# B&R Automation Studio project PT_KB_V01 (part 5)

#### vfdMain.st
```iecst
(* Glavni VFD orchestrator: kontrola, monitoring i dijagnostika po metodi rada. *)
FUNCTION_BLOCK vfdMain

	(* ---------------------------------------------------------------------- *)
	(* 1) Pristup centralnoj VFD strukturi preko prosledjene adrese            *)
	(* ---------------------------------------------------------------------- *)
	vfd_struct_data ACCESS addr_struct;

	(* ---------------------------------------------------------------------- *)
	(* 2) METOD_ENC_CANOPEN                                                     *)
	(* ---------------------------------------------------------------------- *)
	IF vfd_struct_data.settings.METOD_OF_CONTROL = METOD_ENC_CANOPEN THEN

		vfd_struct_data.status.act_power := UINT_TO_REAL(vfd_struct_data.mapping.CanOpen.r_power)/10.0;
		vfd_struct_data.status.act_current := UINT_TO_REAL(vfd_struct_data.mapping.CanOpen.r_current)/100.0;
		vfd_struct_data.status.act_torque := UINT_TO_REAL(vfd_struct_data.mapping.CanOpen.r_torque);
		vfd_struct_data.status.act_freq := UINT_TO_REAL(vfd_struct_data.mapping.CanOpen.r_freq)/100.0;
		vfd_struct_data.status.act_voltage := UINT_TO_REAL(vfd_struct_data.mapping.CanOpen.r_voltage);
		vfd_struct_data.status.act_velocity := UINT_TO_REAL(vfd_struct_data.mapping.CanOpen.r_velocity);

		IF vfd_struct_data.params.Freq > 100.0 THEN
			vfd_struct_data.params.Freq := 100.0;
		END_IF

		(* Skaliranje procentualnog zahteva frekvencije u raw CANopen opseg. *)
		vfd_struct_data.mapping.CanOpen.w_freq := REAL_TO_UINT((((vfd_struct_data.settings.MAX_Freq - vfd_struct_data.settings.MIN_Freq)/100.0)*vfd_struct_data.params.Freq - vfd_struct_data.settings.MIN_Freq)*100.0);
		vfd_struct_data.mapping.CanOpen.w_acc := REAL_TO_UINT(vfd_struct_data.params.Acc*10.0);
		vfd_struct_data.mapping.CanOpen.w_dec := REAL_TO_UINT(vfd_struct_data.params.Dec*10.0);

		fControlENC.cmd := vfd_struct_data.cmds;
		fControlENC.in_addr_CtrlWord := ADR(vfd_struct_data.mapping.CanOpen.CtrlWord);
		fControlENC.in_addr_StatusWord := ADR(vfd_struct_data.mapping.CanOpen.StatusWord);
		fControlENC.in_addr_r_CtrlWord := ADR(vfd_struct_data.mapping.CanOpen.r_CtrlWord);
		fControlENC();

		fStateENC.in_addr_StatusWord := ADR(vfd_struct_data.mapping.CanOpen.StatusWord);
		fStateENC();
		vfd_struct_data.states.state_word := fStateENC.out_State;

		IF NOT(vfd_struct_data.cmds.Enable) THEN
			state_case := ST_PWR_OFF;
		ELSE
			state_case := vfd_struct_data.states.state_word;
		END_IF;

		IF (vfd_struct_data.settings.HaveOverCurrentProtection) AND NOT(vfd_struct_data.mapping.CanOpenATV.r_OverCurrentProtect) THEN
			state_case := ST_CURRPROTECT;
			vfd_struct_data.states.OVERCURRENT_PROTECT := TRUE;
		ELSE
			vfd_struct_data.states.OVERCURRENT_PROTECT := FALSE;
		END_IF;

		Done := fControlENC.out_DONE;
		Busy := fControlENC.out_BUSY;
		errorID := vfd_struct_data.mapping.CanOpen.r_errorCode;

		(* Mapiranje internog state_case u bool state izlaze za HMI/SCADA. *)
		CASE state_case OF
			ST_PWR_OFF:
				vfd_struct_data.states.PWR_ON := FALSE;
				vfd_struct_data.states.READY := FALSE;
				vfd_struct_data.states.PREOPERATIONAL := FALSE;
				vfd_struct_data.states.RUN := FALSE;
				vfd_struct_data.states.STOPPING := FALSE;
				vfd_struct_data.states.STOPED := FALSE;
				vfd_struct_data.states.FAULT := FALSE;
				vfd_struct_data.states.ALARM := FALSE;
				vfd_struct_data.states.TUNING := FALSE;
				vfd_struct_data.states.JOG := FALSE;
			ST_READY:
				vfd_struct_data.states.PWR_ON := TRUE;
				vfd_struct_data.states.READY := TRUE;
				vfd_struct_data.states.PREOPERATIONAL := FALSE;
				vfd_struct_data.states.RUN := FALSE;
				vfd_struct_data.states.STOPPING := FALSE;
				vfd_struct_data.states.STOPED := FALSE;
				vfd_struct_data.states.FAULT := FALSE;
				vfd_struct_data.states.ALARM := FALSE;
				vfd_struct_data.states.TUNING := FALSE;
				vfd_struct_data.states.JOG := FALSE;
			ST_PREOPERATIONAL:
				vfd_struct_data.states.PWR_ON := TRUE;
				vfd_struct_data.states.READY := FALSE;
				vfd_struct_data.states.PREOPERATIONAL := TRUE;
				vfd_struct_data.states.RUN := FALSE;
				vfd_struct_data.states.STOPPING := FALSE;
				vfd_struct_data.states.STOPED := FALSE;
				vfd_struct_data.states.FAULT := FALSE;
				vfd_struct_data.states.ALARM := FALSE;
				vfd_struct_data.states.TUNING := FALSE;
				vfd_struct_data.states.JOG := FALSE;
			ST_RUN:
				vfd_struct_data.states.PWR_ON := TRUE;
				vfd_struct_data.states.READY := FALSE;
				vfd_struct_data.states.PREOPERATIONAL := FALSE;
				vfd_struct_data.states.RUN := TRUE;
				vfd_struct_data.states.STOPPING := FALSE;
				vfd_struct_data.states.STOPED := FALSE;
				vfd_struct_data.states.FAULT := FALSE;
				vfd_struct_data.states.ALARM := FALSE;
				vfd_struct_data.states.TUNING := FALSE;
				vfd_struct_data.states.JOG := FALSE;
			ST_STOPPING:
				vfd_struct_data.states.PWR_ON := TRUE;
				vfd_struct_data.states.READY := FALSE;
				vfd_struct_data.states.PREOPERATIONAL := FALSE;
				vfd_struct_data.states.RUN := FALSE;
				vfd_struct_data.states.STOPPING := TRUE;
				vfd_struct_data.states.STOPED := FALSE;
				vfd_struct_data.states.FAULT := FALSE;
				vfd_struct_data.states.ALARM := FALSE;
				vfd_struct_data.states.TUNING := FALSE;
				vfd_struct_data.states.JOG := FALSE;
			ST_STOPPED:
				vfd_struct_data.states.PWR_ON := TRUE;
				vfd_struct_data.states.READY := FALSE;
				vfd_struct_data.states.PREOPERATIONAL := FALSE;
				vfd_struct_data.states.RUN := FALSE;
				vfd_struct_data.states.STOPPING := FALSE;
				vfd_struct_data.states.STOPED := TRUE;
				vfd_struct_data.states.FAULT := FALSE;
				vfd_struct_data.states.ALARM := FALSE;
				vfd_struct_data.states.TUNING := FALSE;
				vfd_struct_data.states.JOG := FALSE;
			ST_FAULT:
				vfd_struct_data.states.PWR_ON := FALSE;
				vfd_struct_data.states.READY := FALSE;
				vfd_struct_data.states.PREOPERATIONAL := FALSE;
				vfd_struct_data.states.RUN := FALSE;
				vfd_struct_data.states.STOPPING := FALSE;
				vfd_struct_data.states.STOPED := FALSE;
				vfd_struct_data.states.FAULT := TRUE;
				vfd_struct_data.states.ALARM := FALSE;
				vfd_struct_data.states.TUNING := FALSE;
				vfd_struct_data.states.JOG := FALSE;
			ST_ALARM:
				vfd_struct_data.states.PWR_ON := TRUE;
				vfd_struct_data.states.READY := FALSE;
				vfd_struct_data.states.PREOPERATIONAL := FALSE;
				vfd_struct_data.states.RUN := FALSE;
				vfd_struct_data.states.STOPPING := FALSE;
				vfd_struct_data.states.STOPED := FALSE;
				vfd_struct_data.states.FAULT := FALSE;
				vfd_struct_data.states.ALARM := TRUE;
				vfd_struct_data.states.TUNING := FALSE;
				vfd_struct_data.states.JOG := FALSE;
			ST_TUNING:
				vfd_struct_data.states.PWR_ON := TRUE;
				vfd_struct_data.states.READY := FALSE;
				vfd_struct_data.states.PREOPERATIONAL := FALSE;
				vfd_struct_data.states.RUN := FALSE;
				vfd_struct_data.states.STOPPING := FALSE;
				vfd_struct_data.states.STOPED := FALSE;
				vfd_struct_data.states.FAULT := FALSE;
				vfd_struct_data.states.ALARM := FALSE;
				vfd_struct_data.states.TUNING := TRUE;
				vfd_struct_data.states.JOG := FALSE;
			ST_JOG:
				vfd_struct_data.states.PWR_ON := TRUE;
				vfd_struct_data.states.READY := FALSE;
				vfd_struct_data.states.PREOPERATIONAL := FALSE;
				vfd_struct_data.states.RUN := FALSE;
				vfd_struct_data.states.STOPPING := FALSE;
				vfd_struct_data.states.STOPED := FALSE;
				vfd_struct_data.states.FAULT := FALSE;
				vfd_struct_data.states.ALARM := FALSE;
				vfd_struct_data.states.TUNING := FALSE;
				vfd_struct_data.states.JOG := TRUE;
			ST_CURRPROTECT:
				vfd_struct_data.states.PWR_ON := FALSE;
				vfd_struct_data.states.READY := FALSE;
				vfd_struct_data.states.PREOPERATIONAL := FALSE;
				vfd_struct_data.states.RUN := FALSE;
				vfd_struct_data.states.STOPPING := FALSE;
				vfd_struct_data.states.STOPED := FALSE;
				vfd_struct_data.states.FAULT := FALSE;
				vfd_struct_data.states.ALARM := FALSE;
				vfd_struct_data.states.TUNING := FALSE;
				vfd_struct_data.states.JOG := FALSE;
				vfd_struct_data.states.OVERCURRENT_PROTECT := TRUE;
			ELSE
				vfd_struct_data.states.PWR_ON := TRUE;
				vfd_struct_data.states.READY := FALSE;
				vfd_struct_data.states.PREOPERATIONAL := FALSE;
				vfd_struct_data.states.RUN := FALSE;
				vfd_struct_data.states.STOPPING := FALSE;
				vfd_struct_data.states.STOPED := FALSE;
				vfd_struct_data.states.FAULT := FALSE;
				vfd_struct_data.states.ALARM := FALSE;
				vfd_struct_data.states.TUNING := FALSE;
				vfd_struct_data.states.JOG := FALSE;
		END_CASE;

	END_IF;

	(* ---------------------------------------------------------------------- *)
	(* 3) METOD_DIO                                                             *)
	(* ---------------------------------------------------------------------- *)
	IF vfd_struct_data.settings.METOD_OF_CONTROL = METOD_DIO THEN

		IF vfd_struct_data.cmds.Enable THEN

			(* Legacy ekvivalent skale: REAL_TO_INT((Freq)*32767.0/100.0). *)
			IF vfd_struct_data.params.Freq > 100.0 THEN
				vfd_struct_data.params.Freq := 100.0;
			END_IF

			vfd_struct_data.mapping.DIO.w_freq := REAL_TO_INT((32767.0/100.0)*vfd_struct_data.params.Freq);
			vfd_struct_data.mapping.DIO.w_run_fwd := vfd_struct_data.cmds.Run_fwd;
			vfd_struct_data.mapping.DIO.w_run_rev := vfd_struct_data.cmds.Run_rev;
			vfd_struct_data.mapping.DIO.w_jog_fwd := vfd_struct_data.cmds.Jog_fwd;
			vfd_struct_data.mapping.DIO.w_jog_rev := vfd_struct_data.cmds.Jog_rev;
			vfd_struct_data.mapping.DIO.w_Stop := vfd_struct_data.cmds.Stop;
			vfd_struct_data.mapping.DIO.w_faststop := vfd_struct_data.cmds.FastStop;

			vfd_struct_data.status.act_freq := (((vfd_struct_data.settings.MAX_Freq - vfd_struct_data.settings.MIN_Freq)/32767.0)*vfd_struct_data.mapping.DIO.r_freq - vfd_struct_data.settings.MIN_Freq)*100.0;

			(* Legacy ekvivalent citanja: REAL_TO_UINT((r_freq)*100.0/32767.0). *)
			state_case := ST_READY;
		ELSE
			vfd_struct_data.mapping.DIO.w_freq := 0;
			vfd_struct_data.mapping.DIO.w_run_fwd := FALSE;
			vfd_struct_data.mapping.DIO.w_run_rev := FALSE;
			vfd_struct_data.mapping.DIO.w_jog_fwd := FALSE;
			vfd_struct_data.mapping.DIO.w_jog_rev := FALSE;
			vfd_struct_data.mapping.DIO.w_Stop := FALSE;
			vfd_struct_data.mapping.DIO.w_faststop := FALSE;
			state_case := ST_PWR_OFF;
		END_IF

			vfd_struct_data.mapping.DIO.w_reset := vfd_struct_data.cmds.Reset;
		   IF NOT (vfd_struct_data.mapping.DIO.r_error) THEN
			   state_case := ST_FAULT;
		   END_IF

		IF (vfd_struct_data.settings.HaveOverCurrentProtection) AND NOT(vfd_struct_data.mapping.CanOpenATV.r_OverCurrentProtect) THEN
			state_case := ST_CURRPROTECT;
			vfd_struct_data.states.OVERCURRENT_PROTECT := TRUE;
		ELSE
			vfd_struct_data.states.OVERCURRENT_PROTECT := FALSE;
		END_IF;

		(* U DIO metodi koristi se isti izlazni model states.*)
		CASE state_case OF
			ST_PWR_OFF:
				vfd_struct_data.states.PWR_ON := FALSE;
				vfd_struct_data.states.READY := FALSE;
				vfd_struct_data.states.PREOPERATIONAL := FALSE;
				vfd_struct_data.states.RUN := FALSE;
				vfd_struct_data.states.STOPPING := FALSE;
				vfd_struct_data.states.STOPED := FALSE;
				vfd_struct_data.states.FAULT := FALSE;
				vfd_struct_data.states.ALARM := FALSE;
				vfd_struct_data.states.TUNING := FALSE;
				vfd_struct_data.states.JOG := FALSE;
			ST_READY:
				vfd_struct_data.states.PWR_ON := TRUE;
				vfd_struct_data.states.READY := TRUE;
				vfd_struct_data.states.PREOPERATIONAL := FALSE;
				vfd_struct_data.states.RUN := FALSE;
				vfd_struct_data.states.STOPPING := FALSE;
				vfd_struct_data.states.STOPED := FALSE;
				vfd_struct_data.states.FAULT := FALSE;
				vfd_struct_data.states.ALARM := FALSE;
				vfd_struct_data.states.TUNING := FALSE;
				vfd_struct_data.states.JOG := FALSE;
			ST_PREOPERATIONAL:
				vfd_struct_data.states.PWR_ON := TRUE;
				vfd_struct_data.states.READY := FALSE;
				vfd_struct_data.states.PREOPERATIONAL := TRUE;
				vfd_struct_data.states.RUN := FALSE;
				vfd_struct_data.states.STOPPING := FALSE;
				vfd_struct_data.states.STOPED := FALSE;
				vfd_struct_data.states.FAULT := FALSE;
				vfd_struct_data.states.ALARM := FALSE;
				vfd_struct_data.states.TUNING := FALSE;
				vfd_struct_data.states.JOG := FALSE;
			ST_RUN:
				vfd_struct_data.states.PWR_ON := TRUE;
				vfd_struct_data.states.READY := FALSE;
				vfd_struct_data.states.PREOPERATIONAL := FALSE;
				vfd_struct_data.states.RUN := TRUE;
				vfd_struct_data.states.STOPPING := FALSE;
				vfd_struct_data.states.STOPED := FALSE;
				vfd_struct_data.states.FAULT := FALSE;
				vfd_struct_data.states.ALARM := FALSE;
				vfd_struct_data.states.TUNING := FALSE;
				vfd_struct_data.states.JOG := FALSE;
			ST_STOPPING:
				vfd_struct_data.states.PWR_ON := TRUE;
				vfd_struct_data.states.READY := FALSE;
				vfd_struct_data.states.PREOPERATIONAL := FALSE;
				vfd_struct_data.states.RUN := FALSE;
				vfd_struct_data.states.STOPPING := TRUE;
				vfd_struct_data.states.STOPED := FALSE;
				vfd_struct_data.states.FAULT := FALSE;
				vfd_struct_data.states.ALARM := FALSE;
				vfd_struct_data.states.TUNING := FALSE;
				vfd_struct_data.states.JOG := FALSE;
			ST_STOPPED:
				vfd_struct_data.states.PWR_ON := TRUE;
				vfd_struct_data.states.READY := FALSE;
				vfd_struct_data.states.PREOPERATIONAL := FALSE;
				vfd_struct_data.states.RUN := FALSE;
				vfd_struct_data.states.STOPPING := FALSE;
				vfd_struct_data.states.STOPED := TRUE;
				vfd_struct_data.states.FAULT := FALSE;
				vfd_struct_data.states.ALARM := FALSE;
				vfd_struct_data.states.TUNING := FALSE;
				vfd_struct_data.states.JOG := FALSE;
			ST_FAULT:
				vfd_struct_data.states.PWR_ON := FALSE;
				vfd_struct_data.states.READY := FALSE;
				vfd_struct_data.states.PREOPERATIONAL := FALSE;
				vfd_struct_data.states.RUN := FALSE;
				vfd_struct_data.states.STOPPING := FALSE;
				vfd_struct_data.states.STOPED := FALSE;
				vfd_struct_data.states.FAULT := TRUE;
				vfd_struct_data.states.ALARM := FALSE;
				vfd_struct_data.states.TUNING := FALSE;
				vfd_struct_data.states.JOG := FALSE;
			ST_ALARM:
				vfd_struct_data.states.PWR_ON := TRUE;
				vfd_struct_data.states.READY := FALSE;
				vfd_struct_data.states.PREOPERATIONAL := FALSE;
				vfd_struct_data.states.RUN := FALSE;
				vfd_struct_data.states.STOPPING := FALSE;
				vfd_struct_data.states.STOPED := FALSE;
				vfd_struct_data.states.FAULT := FALSE;
				vfd_struct_data.states.ALARM := TRUE;
				vfd_struct_data.states.TUNING := FALSE;
				vfd_struct_data.states.JOG := FALSE;
			ST_TUNING:
				vfd_struct_data.states.PWR_ON := TRUE;
				vfd_struct_data.states.READY := FALSE;
				vfd_struct_data.states.PREOPERATIONAL := FALSE;
				vfd_struct_data.states.RUN := FALSE;
				vfd_struct_data.states.STOPPING := FALSE;
				vfd_struct_data.states.STOPED := FALSE;
				vfd_struct_data.states.FAULT := FALSE;
				vfd_struct_data.states.ALARM := FALSE;
				vfd_struct_data.states.TUNING := TRUE;
				vfd_struct_data.states.JOG := FALSE;
			ST_JOG:
				vfd_struct_data.states.PWR_ON := TRUE;
				vfd_struct_data.states.READY := FALSE;
				vfd_struct_data.states.PREOPERATIONAL := FALSE;
				vfd_struct_data.states.RUN := FALSE;
				vfd_struct_data.states.STOPPING := FALSE;
				vfd_struct_data.states.STOPED := FALSE;
				vfd_struct_data.states.FAULT := FALSE;
				vfd_struct_data.states.ALARM := FALSE;
				vfd_struct_data.states.TUNING := FALSE;
				vfd_struct_data.states.JOG := TRUE;
			ST_CURRPROTECT:
				vfd_struct_data.states.PWR_ON := FALSE;
				vfd_struct_data.states.READY := FALSE;
				vfd_struct_data.states.PREOPERATIONAL := FALSE;
				vfd_struct_data.states.RUN := FALSE;
				vfd_struct_data.states.STOPPING := FALSE;
				vfd_struct_data.states.STOPED := FALSE;
				vfd_struct_data.states.FAULT := FALSE;
				vfd_struct_data.states.ALARM := FALSE;
				vfd_struct_data.states.TUNING := FALSE;
				vfd_struct_data.states.JOG := FALSE;
				vfd_struct_data.states.OVERCURRENT_PROTECT := TRUE;
			ELSE
				vfd_struct_data.states.PWR_ON := TRUE;
				vfd_struct_data.states.READY := FALSE;
				vfd_struct_data.states.PREOPERATIONAL := FALSE;
				vfd_struct_data.states.RUN := FALSE;
				vfd_struct_data.states.STOPPING := FALSE;
				vfd_struct_data.states.STOPED := FALSE;
				vfd_struct_data.states.FAULT := FALSE;
				vfd_struct_data.states.ALARM := FALSE;
				vfd_struct_data.states.TUNING := FALSE;
				vfd_struct_data.states.JOG := FALSE;
		END_CASE;

	END_IF;

	(* ---------------------------------------------------------------------- *)
	(* 4) METOD_DIO_CANOPEN                                                     *)
	(* ---------------------------------------------------------------------- *)
	IF vfd_struct_data.settings.METOD_OF_CONTROL = METOD_DIO_CANOPEN THEN

		IF vfd_struct_data.cmds.Enable THEN

			IF vfd_struct_data.params.Freq > 100.0 THEN
				vfd_struct_data.params.Freq := 100.0;
			END_IF

			vfd_struct_data.mapping.DIO.w_freq := REAL_TO_INT((32767.0/100.0)*vfd_struct_data.params.Freq);

			(* Legacy alternativa skale (ne koristi se u aktivnoj logici). *)
			vfd_struct_data.mapping.DIO.w_run_fwd := vfd_struct_data.cmds.Run_fwd;
			vfd_struct_data.mapping.DIO.w_run_rev := vfd_struct_data.cmds.Run_rev;
			vfd_struct_data.mapping.DIO.w_jog_fwd := vfd_struct_data.cmds.Jog_fwd;
			vfd_struct_data.mapping.DIO.w_jog_rev := vfd_struct_data.cmds.Jog_rev;
			vfd_struct_data.mapping.DIO.w_Stop := vfd_struct_data.cmds.Stop;
			vfd_struct_data.mapping.DIO.w_faststop := vfd_struct_data.cmds.FastStop;
			(* Legacy ekvivalent citanja: REAL_TO_UINT((r_freq)*100.0/32767.0). *)
		ELSE
			vfd_struct_data.mapping.DIO.w_freq := 0;
			vfd_struct_data.mapping.DIO.w_run_fwd := FALSE;
			vfd_struct_data.mapping.DIO.w_run_rev := FALSE;
			vfd_struct_data.mapping.DIO.w_jog_fwd := FALSE;
			vfd_struct_data.mapping.DIO.w_jog_rev := FALSE;
			vfd_struct_data.mapping.DIO.w_Stop := FALSE;
			vfd_struct_data.mapping.DIO.w_faststop := FALSE;

		END_IF

		vfd_struct_data.mapping.DIO.w_reset := vfd_struct_data.cmds.Reset;

		vfd_struct_data.status.act_power := UINT_TO_REAL(vfd_struct_data.mapping.CanOpen.r_power)/10.0;
		vfd_struct_data.status.act_current := UINT_TO_REAL(vfd_struct_data.mapping.CanOpen.r_current)/100.0;
		vfd_struct_data.status.act_torque := UINT_TO_REAL(vfd_struct_data.mapping.CanOpen.r_torque);
		vfd_struct_data.status.act_freq := UINT_TO_REAL(vfd_struct_data.mapping.CanOpen.r_freq)/100.0;
		vfd_struct_data.status.act_voltage := UINT_TO_REAL(vfd_struct_data.mapping.CanOpen.r_voltage);
		vfd_struct_data.status.act_velocity := UINT_TO_REAL(vfd_struct_data.mapping.CanOpen.r_velocity);

		vfd_struct_data.mapping.CanOpen.w_acc := REAL_TO_UINT(vfd_struct_data.params.Acc*10.0);
		vfd_struct_data.mapping.CanOpen.w_dec := REAL_TO_UINT(vfd_struct_data.params.Dec*10.0);

		fStateENC.in_addr_StatusWord := ADR(vfd_struct_data.mapping.CanOpen.StatusWord);
		fStateENC();
		vfd_struct_data.states.state_word := fStateENC.out_State;

		IF NOT(vfd_struct_data.cmds.Enable) THEN
			state_case := ST_PWR_OFF;
		ELSE
			state_case := vfd_struct_data.states.state_word;
		END_IF;

		IF (vfd_struct_data.settings.HaveOverCurrentProtection) AND NOT(vfd_struct_data.mapping.CanOpenATV.r_OverCurrentProtect) THEN
			state_case := ST_CURRPROTECT;
			vfd_struct_data.states.OVERCURRENT_PROTECT := TRUE;
		ELSE
			vfd_struct_data.states.OVERCURRENT_PROTECT := FALSE;
		END_IF;

		(* U kombinovanoj metodi Done/Busy se ne preuzimaju iz ENC control FB-a. *)
		errorID := vfd_struct_data.mapping.CanOpen.r_errorCode;

		(* Kombinovana metoda: komande kroz DIO, status kroz CANopen. *)
		CASE state_case OF
			ST_PWR_OFF:
				vfd_struct_data.states.PWR_ON := FALSE;
				vfd_struct_data.states.READY := FALSE;
				vfd_struct_data.states.PREOPERATIONAL := FALSE;
				vfd_struct_data.states.RUN := FALSE;
				vfd_struct_data.states.STOPPING := FALSE;
				vfd_struct_data.states.STOPED := FALSE;
				vfd_struct_data.states.FAULT := FALSE;
				vfd_struct_data.states.ALARM := FALSE;
				vfd_struct_data.states.TUNING := FALSE;
				vfd_struct_data.states.JOG := FALSE;
			ST_READY:
				vfd_struct_data.states.PWR_ON := TRUE;
				vfd_struct_data.states.READY := TRUE;
				vfd_struct_data.states.PREOPERATIONAL := FALSE;
				vfd_struct_data.states.RUN := FALSE;
				vfd_struct_data.states.STOPPING := FALSE;
				vfd_struct_data.states.STOPED := FALSE;
				vfd_struct_data.states.FAULT := FALSE;
				vfd_struct_data.states.ALARM := FALSE;
				vfd_struct_data.states.TUNING := FALSE;
				vfd_struct_data.states.JOG := FALSE;
			ST_PREOPERATIONAL:
				vfd_struct_data.states.PWR_ON := TRUE;
				vfd_struct_data.states.READY := FALSE;
				vfd_struct_data.states.PREOPERATIONAL := TRUE;
				vfd_struct_data.states.RUN := FALSE;
				vfd_struct_data.states.STOPPING := FALSE;
				vfd_struct_data.states.STOPED := FALSE;
				vfd_struct_data.states.FAULT := FALSE;
				vfd_struct_data.states.ALARM := FALSE;
				vfd_struct_data.states.TUNING := FALSE;
				vfd_struct_data.states.JOG := FALSE;
			ST_RUN:
				vfd_struct_data.states.PWR_ON := TRUE;
				vfd_struct_data.states.READY := FALSE;
				vfd_struct_data.states.PREOPERATIONAL := FALSE;
				vfd_struct_data.states.RUN := TRUE;
				vfd_struct_data.states.STOPPING := FALSE;
				vfd_struct_data.states.STOPED := FALSE;
				vfd_struct_data.states.FAULT := FALSE;
				vfd_struct_data.states.ALARM := FALSE;
				vfd_struct_data.states.TUNING := FALSE;
				vfd_struct_data.states.JOG := FALSE;
			ST_STOPPING:
				vfd_struct_data.states.PWR_ON := TRUE;
				vfd_struct_data.states.READY := FALSE;
				vfd_struct_data.states.PREOPERATIONAL := FALSE;
				vfd_struct_data.states.RUN := FALSE;
				vfd_struct_data.states.STOPPING := TRUE;
				vfd_struct_data.states.STOPED := FALSE;
				vfd_struct_data.states.FAULT := FALSE;
				vfd_struct_data.states.ALARM := FALSE;
				vfd_struct_data.states.TUNING := FALSE;
				vfd_struct_data.states.JOG := FALSE;
			ST_STOPPED:
				vfd_struct_data.states.PWR_ON := TRUE;
				vfd_struct_data.states.READY := FALSE;
				vfd_struct_data.states.PREOPERATIONAL := FALSE;
				vfd_struct_data.states.RUN := FALSE;
				vfd_struct_data.states.STOPPING := FALSE;
				vfd_struct_data.states.STOPED := TRUE;
				vfd_struct_data.states.FAULT := FALSE;
				vfd_struct_data.states.ALARM := FALSE;
				vfd_struct_data.states.TUNING := FALSE;
				vfd_struct_data.states.JOG := FALSE;
			ST_FAULT:
				vfd_struct_data.states.PWR_ON := FALSE;
				vfd_struct_data.states.READY := FALSE;
				vfd_struct_data.states.PREOPERATIONAL := FALSE;
				vfd_struct_data.states.RUN := FALSE;
				vfd_struct_data.states.STOPPING := FALSE;
				vfd_struct_data.states.STOPED := FALSE;
				vfd_struct_data.states.FAULT := TRUE;
				vfd_struct_data.states.ALARM := FALSE;
				vfd_struct_data.states.TUNING := FALSE;
				vfd_struct_data.states.JOG := FALSE;
			ST_ALARM:
				vfd_struct_data.states.PWR_ON := TRUE;
				vfd_struct_data.states.READY := FALSE;
				vfd_struct_data.states.PREOPERATIONAL := FALSE;
				vfd_struct_data.states.RUN := FALSE;
				vfd_struct_data.states.STOPPING := FALSE;
				vfd_struct_data.states.STOPED := FALSE;
				vfd_struct_data.states.FAULT := FALSE;
				vfd_struct_data.states.ALARM := TRUE;
				vfd_struct_data.states.TUNING := FALSE;
				vfd_struct_data.states.JOG := FALSE;
			ST_TUNING:
				vfd_struct_data.states.PWR_ON := TRUE;
				vfd_struct_data.states.READY := FALSE;
				vfd_struct_data.states.PREOPERATIONAL := FALSE;
				vfd_struct_data.states.RUN := FALSE;
				vfd_struct_data.states.STOPPING := FALSE;
				vfd_struct_data.states.STOPED := FALSE;
				vfd_struct_data.states.FAULT := FALSE;
				vfd_struct_data.states.ALARM := FALSE;
				vfd_struct_data.states.TUNING := TRUE;
				vfd_struct_data.states.JOG := FALSE;
			ST_JOG:
				vfd_struct_data.states.PWR_ON := TRUE;
				vfd_struct_data.states.READY := FALSE;
				vfd_struct_data.states.PREOPERATIONAL := FALSE;
				vfd_struct_data.states.RUN := FALSE;
				vfd_struct_data.states.STOPPING := FALSE;
				vfd_struct_data.states.STOPED := FALSE;
				vfd_struct_data.states.FAULT := FALSE;
				vfd_struct_data.states.ALARM := FALSE;
				vfd_struct_data.states.TUNING := FALSE;
				vfd_struct_data.states.JOG := TRUE;
			ST_CURRPROTECT:
				vfd_struct_data.states.PWR_ON := FALSE;
				vfd_struct_data.states.READY := FALSE;
				vfd_struct_data.states.PREOPERATIONAL := FALSE;
				vfd_struct_data.states.RUN := FALSE;
				vfd_struct_data.states.STOPPING := FALSE;
				vfd_struct_data.states.STOPED := FALSE;
				vfd_struct_data.states.FAULT := FALSE;
				vfd_struct_data.states.ALARM := FALSE;
				vfd_struct_data.states.TUNING := FALSE;
				vfd_struct_data.states.JOG := FALSE;
				vfd_struct_data.states.OVERCURRENT_PROTECT := TRUE;
			ELSE
				vfd_struct_data.states.PWR_ON := TRUE;
				vfd_struct_data.states.READY := FALSE;
				vfd_struct_data.states.PREOPERATIONAL := FALSE;
				vfd_struct_data.states.RUN := FALSE;
				vfd_struct_data.states.STOPPING := FALSE;
				vfd_struct_data.states.STOPED := FALSE;
				vfd_struct_data.states.FAULT := FALSE;
				vfd_struct_data.states.ALARM := FALSE;
				vfd_struct_data.states.TUNING := FALSE;
				vfd_struct_data.states.JOG := FALSE;
		END_CASE;

	END_IF;

	(* ---------------------------------------------------------------------- *)
	(* 5) METOD_ATV_CANOPEN                                                     *)
	(* ---------------------------------------------------------------------- *)
	IF vfd_struct_data.settings.METOD_OF_CONTROL = METOD_ATV_CANOPEN THEN

		vfd_struct_data.status.act_power := INT_TO_REAL(vfd_struct_data.mapping.CanOpenATV.r_power)*vfd_struct_data.settings.RatedMotorPower/100.0;
		vfd_struct_data.status.act_current := UINT_TO_REAL(vfd_struct_data.mapping.CanOpenATV.r_current)/10.0;
		vfd_struct_data.status.act_torque := INT_TO_REAL(vfd_struct_data.mapping.CanOpenATV.r_torque);
		vfd_struct_data.status.act_freq := INT_TO_REAL(vfd_struct_data.mapping.CanOpenATV.r_freq)/100.0;
		vfd_struct_data.status.act_voltage := UINT_TO_REAL(vfd_struct_data.mapping.CanOpenATV.r_voltage);
		vfd_struct_data.status.act_velocity := INT_TO_REAL(vfd_struct_data.mapping.CanOpenATV.ControlEffort);

		vfd_struct_data.mapping.CanOpenATV.w_acc := REAL_TO_UINT(vfd_struct_data.params.Acc*10.0);
		vfd_struct_data.mapping.CanOpenATV.w_dec := REAL_TO_UINT(vfd_struct_data.params.Dec*10.0);

		fStateATV.in_addr_StatusWord := ADR(vfd_struct_data.mapping.CanOpenATV.StatusWord);
		fStateATV();
		vfd_struct_data.states.state_word := fStateATV.out_State;

		fControlATV.cmd := vfd_struct_data.cmds;
		fControlATV.in_addr_CtrlWord := ADR(vfd_struct_data.mapping.CanOpenATV.CtrlWord);
		fControlATV.DC_BUS_STATE := fStateATV.DC_BUS_ON;
		fControlATV.StatusWord := fStateATV.out_State;

		IF vfd_struct_data.params.Freq > 100.0 THEN
			vfd_struct_data.params.Freq := 100.0;
		END_IF

		(* Konverzija procentualnog SP u ATV velocity zahtev. *)
		fControlATV.in_set_freq := REAL_TO_INT(vfd_struct_data.params.Freq*(vfd_struct_data.settings.MAX_Velocity)/100.0);

		fControlATV();
		vfd_struct_data.mapping.CanOpenATV.w_TargetVelocity := fControlATV.set_freq;

		IF NOT(vfd_struct_data.cmds.Enable) THEN
			state_case := STATV_PWR_OFF;
		ELSE
			state_case := vfd_struct_data.states.state_word;
		END_IF;

		IF (vfd_struct_data.settings.HaveOverCurrentProtection) AND NOT(vfd_struct_data.mapping.CanOpenATV.r_OverCurrentProtect) THEN
			state_case := STATV_OVR_CURR;
			vfd_struct_data.states.OVERCURRENT_PROTECT := TRUE;
		ELSE
			vfd_struct_data.states.OVERCURRENT_PROTECT := FALSE;
		END_IF;

		Done := fControlATV.out_DONE;
		Busy := fControlATV.out_BUSY;
		errorID := vfd_struct_data.mapping.CanOpen.r_errorCode;

		(* ATV-specific state kodovi se mapiraju na zajednicke states bool izlaze. *)
		CASE state_case OF
			STATV_PWR_OFF:
				vfd_struct_data.states.PWR_ON := FALSE;
				vfd_struct_data.states.READY := FALSE;
				vfd_struct_data.states.PREOPERATIONAL := FALSE;
				vfd_struct_data.states.RUN := FALSE;
				vfd_struct_data.states.STOPPING := FALSE;
				vfd_struct_data.states.STOPED := FALSE;
				vfd_struct_data.states.FAULT := FALSE;
				vfd_struct_data.states.ALARM := FALSE;
				vfd_struct_data.states.TUNING := FALSE;
				vfd_struct_data.states.JOG := FALSE;
			STATV_RDY:
				vfd_struct_data.states.PWR_ON := TRUE;
				vfd_struct_data.states.READY := TRUE;
				vfd_struct_data.states.PREOPERATIONAL := FALSE;
				vfd_struct_data.states.RUN := FALSE;
				vfd_struct_data.states.STOPPING := FALSE;
				vfd_struct_data.states.STOPED := FALSE;
				vfd_struct_data.states.FAULT := FALSE;
				vfd_struct_data.states.ALARM := FALSE;
				vfd_struct_data.states.TUNING := FALSE;
				vfd_struct_data.states.JOG := FALSE;
			STATV_SWH_ON:
				vfd_struct_data.states.PWR_ON := TRUE;
				vfd_struct_data.states.READY := FALSE;
				vfd_struct_data.states.PREOPERATIONAL := TRUE;
				vfd_struct_data.states.RUN := FALSE;
				vfd_struct_data.states.STOPPING := FALSE;
				vfd_struct_data.states.STOPED := FALSE;
				vfd_struct_data.states.FAULT := FALSE;
				vfd_struct_data.states.ALARM := FALSE;
				vfd_struct_data.states.TUNING := FALSE;
				vfd_struct_data.states.JOG := FALSE;
			STATV_RUN:
				vfd_struct_data.states.PWR_ON := TRUE;
				vfd_struct_data.states.READY := FALSE;
				vfd_struct_data.states.PREOPERATIONAL := FALSE;
				vfd_struct_data.states.RUN := TRUE;
				vfd_struct_data.states.STOPPING := FALSE;
				vfd_struct_data.states.STOPED := FALSE;
				vfd_struct_data.states.FAULT := FALSE;
				vfd_struct_data.states.ALARM := FALSE;
				vfd_struct_data.states.TUNING := FALSE;
				vfd_struct_data.states.JOG := FALSE;
			STATV_SWH_DISABLE:
				vfd_struct_data.states.PWR_ON := TRUE;
				vfd_struct_data.states.READY := FALSE;
				vfd_struct_data.states.PREOPERATIONAL := FALSE;
				vfd_struct_data.states.RUN := FALSE;
				vfd_struct_data.states.STOPPING := TRUE;
				vfd_struct_data.states.STOPED := FALSE;
				vfd_struct_data.states.FAULT := FALSE;
				vfd_struct_data.states.ALARM := FALSE;
				vfd_struct_data.states.TUNING := FALSE;
				vfd_struct_data.states.JOG := FALSE;
			STATV_FAST_STOP:
				vfd_struct_data.states.PWR_ON := TRUE;
				vfd_struct_data.states.READY := FALSE;
				vfd_struct_data.states.PREOPERATIONAL := FALSE;
				vfd_struct_data.states.RUN := FALSE;
				vfd_struct_data.states.STOPPING := FALSE;
				vfd_struct_data.states.STOPED := TRUE;
				vfd_struct_data.states.FAULT := FALSE;
				vfd_struct_data.states.ALARM := FALSE;
				vfd_struct_data.states.TUNING := FALSE;
				vfd_struct_data.states.JOG := FALSE;
			STATV_ERR:
				vfd_struct_data.states.PWR_ON := FALSE;
				vfd_struct_data.states.READY := FALSE;
				vfd_struct_data.states.PREOPERATIONAL := FALSE;
				vfd_struct_data.states.RUN := FALSE;
				vfd_struct_data.states.STOPPING := FALSE;
				vfd_struct_data.states.STOPED := FALSE;
				vfd_struct_data.states.FAULT := TRUE;
				vfd_struct_data.states.ALARM := FALSE;
				vfd_struct_data.states.TUNING := FALSE;
				vfd_struct_data.states.JOG := FALSE;
			STATV_ERR_MNG:
				vfd_struct_data.states.PWR_ON := TRUE;
				vfd_struct_data.states.READY := FALSE;
				vfd_struct_data.states.PREOPERATIONAL := FALSE;
				vfd_struct_data.states.RUN := FALSE;
				vfd_struct_data.states.STOPPING := FALSE;
				vfd_struct_data.states.STOPED := FALSE;
				vfd_struct_data.states.FAULT := FALSE;
				vfd_struct_data.states.ALARM := TRUE;
				vfd_struct_data.states.TUNING := FALSE;
				vfd_struct_data.states.JOG := FALSE;
			STATV_OVR_CURR:
				vfd_struct_data.states.PWR_ON := FALSE;
				vfd_struct_data.states.READY := FALSE;
				vfd_struct_data.states.PREOPERATIONAL := FALSE;
				vfd_struct_data.states.RUN := FALSE;
				vfd_struct_data.states.STOPPING := FALSE;
				vfd_struct_data.states.STOPED := FALSE;
				vfd_struct_data.states.FAULT := FALSE;
				vfd_struct_data.states.ALARM := TRUE;
				vfd_struct_data.states.TUNING := FALSE;
				vfd_struct_data.states.JOG := FALSE;
				vfd_struct_data.states.OVERCURRENT_PROTECT := TRUE;
			ELSE
				vfd_struct_data.states.PWR_ON := TRUE;
				vfd_struct_data.states.READY := FALSE;
				vfd_struct_data.states.PREOPERATIONAL := FALSE;
				vfd_struct_data.states.RUN := FALSE;
				vfd_struct_data.states.STOPPING := FALSE;
				vfd_struct_data.states.STOPED := FALSE;
				vfd_struct_data.states.FAULT := FALSE;
				vfd_struct_data.states.ALARM := FALSE;
				vfd_struct_data.states.TUNING := FALSE;
				vfd_struct_data.states.JOG := FALSE;
		END_CASE;

	END_IF;

	(* ATV modul status se prepisuje u zajednicki ModuleStatusOK kanal. *)
	IF vfd_struct_data.settings.METOD_OF_CONTROL = METOD_ATV_CANOPEN THEN
		vfd_struct_data.mapping.CanOpen.ModuleStatusOK := vfd_struct_data.mapping.CanOpenATV.ModuleStatusOK;
	END_IF;

	(* ---------------------------------------------------------------------- *)
	(* 6) Error management komunikacije                                         *)
	(* ---------------------------------------------------------------------- *)
	ton_dur.PT := T#60s;
	IF (EDGENEG(vfd_struct_data.mapping.CanOpen.ModuleStatusOK)) THEN
		ton_dur.IN := TRUE;
		vfd_struct_data.errorMgmt.Counter_errors := vfd_struct_data.errorMgmt.Counter_errors + 1;
		acum_time := 0;
	END_IF

	IF (ton_dur.Q) AND NOT(vfd_struct_data.mapping.CanOpen.ModuleStatusOK) THEN
		acum_time := acum_time + ton_dur.PT;
		ton_dur.IN := FALSE;
	ELSIF NOT(vfd_struct_data.mapping.CanOpen.ModuleStatusOK) THEN
		ton_dur.IN := TRUE;
	END_IF;

	IF (ton_dur.IN) AND (vfd_struct_data.mapping.CanOpen.ModuleStatusOK) THEN
		ton_dur.IN := FALSE;
		vfd_struct_data.errorMgmt.Last_Duration := ton_dur.ET + acum_time;
		DTGetTime_1.enable:=TRUE;
		DTGetTime_1();
		vfd_struct_data.errorMgmt.Last_time := DTGetTime_1.DT1;
		DTGetTime_1.enable:=FALSE;
		IF(vfd_struct_data.errorMgmt.Last_Duration > vfd_struct_data.errorMgmt.Max_duration) THEN
			vfd_struct_data.errorMgmt.Max_duration := vfd_struct_data.errorMgmt.Last_Duration;
		END_IF

	END_IF
	ton_dur();
	vfd_struct_data.errorMgmt.StatusOK := vfd_struct_data.mapping.CanOpen.ModuleStatusOK;

END_FUNCTION_BLOCK
```

### Library Logical/Libraries/NashCan1 (IEC)

#### Types.typ - Exported data types
```iecst
TYPE
	CanIn : 	STRUCT
		b_NodeState : BOOL; (*Status Noda CAN uredjaja na mrezi*)
		w_StatusReg : UINT; (*Status registar - statusna recenica*)
		w_MotorStruja : UINT; (*Trenutna struja motora u 0,1A *)
		w_MotorBrz : INT; (*Trenutna brzina motora u obrt/min *)
		w_MotorSnaga : INT; (*Trenutna snaga motora u % *)
	END_STRUCT;
	CanOut : 	STRUCT
		w_ControlReg : UINT; (*Kontrolni registar - kontrolna recenica*)
		w_ZadataBrz : INT; (*Brzina koja se salje na regulator u obrt/min*)
	END_STRUCT;
END_TYPE
```

#### NashCan1.fun - Exported functions and function blocks
```iecst
FUNCTION_BLOCK FbCanAtv (*** 	FB za upravljanje ATV Schneider frekventnim regulatorima preko CanOpena	***)
	VAR_INPUT
		AtvCanIn : CanIn; (*Ulazna struktura u CAN FB iz frekventnog regulatora*)
		w_ZadataBrzHz : REAL; (*Zadata brzina u 0,1Hz *)
		w_FR_min : REAL; (*Zadata minimalna brzina u 0,1Hz *)
		w_FR_max : REAL; (*Zadata maksimalna brzina u 0,1Hz *)
		w_NomSnaga : REAL; (*Zadata nominalna snaga frekventnog u kW *)
		b_Enable : BOOL;
		b_Start : BOOL;
		b_AlarmRst : BOOL;
	END_VAR
	VAR_OUTPUT
		AtvCanOut : CanOut;
		w_MotorStruja : REAL; (*Trenutna struja motora u A *)
		w_MotorBrz : REAL; (*Trenutna broj obrtaja motora prevedena u Hz*)
		w_MotorSnaga : REAL; (*Trenutna snaga motora u kW*)
		b_Alarm_FR : BOOL; (*Alarm frekventnog regulatora*)
		b_Alarm_CAN : BOOL; (*Alarm CAN komunikacije*)
		b_Running : BOOL; (*In run status frekventnog regulatora*)
	END_VAR
	VAR
		b_StatusBit00 : BOOL;
		b_StatusBit01 : BOOL;
		b_StatusBit02 : BOOL;
		b_StatusBit03 : BOOL;
		b_StatusBit04 : BOOL;
		b_StatusBit05 : BOOL;
		b_StatusBit06 : BOOL;
		b_StatusBit07 : BOOL;
		b_StatusDissable : BOOL;
		b_StatusSwitchReady : BOOL;
		b_StatusSwitchOn : BOOL;
	END_VAR
END_FUNCTION_BLOCK
```

#### FbCanAtv.st
```iecst
FUNCTION_BLOCK FbCanAtv
	AtvCanOut.w_ZadataBrz:=REAL_TO_INT(w_ZadataBrzHz*60);	//Brzina se na Atv zadaje u Obrt/min
	(* Provera zadate brzine u opsegu Min-Max *)
	IF w_ZadataBrzHz<w_FR_min THEN AtvCanOut.w_ZadataBrz:= REAL_TO_INT(w_FR_min*60); END_IF
	IF w_ZadataBrzHz>w_FR_max THEN AtvCanOut.w_ZadataBrz:= REAL_TO_INT(w_FR_max*60); END_IF

	w_MotorStruja:= UINT_TO_REAL (AtvCanIn.w_MotorStruja) /10;
	w_MotorBrz:= INT_TO_REAL(AtvCanIn.w_MotorBrz)/60;
	w_MotorSnaga:=w_NomSnaga * (INT_TO_REAL(AtvCanIn.w_MotorSnaga))/100; //AtvCanIn.w_MotorSnaga se prima u %

	b_StatusBit00:=	AtvCanIn.w_StatusReg.0;
	b_StatusBit01:=	AtvCanIn.w_StatusReg.1;
	b_StatusBit02:=	AtvCanIn.w_StatusReg.2;
	b_StatusBit03:=	AtvCanIn.w_StatusReg.3;
	b_StatusBit04:=	AtvCanIn.w_StatusReg.4;
	b_StatusBit05:=	AtvCanIn.w_StatusReg.5;
	b_StatusBit06:=	AtvCanIn.w_StatusReg.6;
	b_StatusBit07:=	AtvCanIn.w_StatusReg.7;

	b_StatusDissable:=		NOT(b_StatusBit00) AND NOT(b_StatusBit01) AND NOT(b_StatusBit02) AND NOT(b_StatusBit03) AND b_StatusBit06;
	b_StatusSwitchReady:=	b_StatusBit00 AND NOT(b_StatusBit01) AND NOT(b_StatusBit02) AND NOT(b_StatusBit03) AND b_StatusBit05 AND NOT(b_StatusBit06);
	b_StatusSwitchOn:=		b_StatusBit00 AND b_StatusBit01 AND NOT(b_StatusBit02) AND NOT(b_StatusBit03) AND b_StatusBit05 AND NOT(b_StatusBit06);
	b_Alarm_CAN:=			NOT(AtvCanIn.b_NodeState);
	b_Alarm_FR:=			b_StatusBit03 AND b_Enable;
	b_Running:=				b_StatusBit00 AND b_StatusBit01 AND b_StatusBit02 AND NOT(b_StatusBit03) AND b_StatusBit05 AND NOT(b_StatusBit06);

	IF b_Enable AND NOT(b_StatusSwitchOn) THEN
		IF b_StatusDissable THEN AtvCanOut.w_ControlReg:=6; END_IF //Prebacivanje Atv u stanje SwitchReady
		IF b_StatusSwitchReady THEN AtvCanOut.w_ControlReg:=7; END_IF //Prebacivanje Atv u stanje SwitchOn
	END_IF
	AtvCanOut.w_ControlReg.3:= b_Enable AND b_Start AND (b_StatusSwitchOn OR b_Running);
	//IF NOT(b_Enable) OR b_Alarm_CAN OR b_Alarm_FR THEN AtvCanOut.w_ControlReg:=0; END_IF
	IF NOT(b_Enable) THEN AtvCanOut.w_ControlReg:=0; END_IF
	AtvCanOut.w_ControlReg.7:=b_AlarmRst;
END_FUNCTION_BLOCK
```

- Visualisation Logical/Visu1 (not shown)

### Program Logical/IO (IEC)

#### Cyclic.st
```iecst
PROGRAM _CYCLIC

(* ============================================================================ *)
(* IO_CYCLIC  Pozivi svih BR_Lib FB instanci                                   *)
(* Objekat: PG  Podstanica grejanja 1, Kursumlijska Banja                     *)
(* Sva IO mapiranja su u IoMap.iom  ovde su samo pozivi FB-ova.               *)
(* Redosled: senzori -> DI -> AV -> RV -> PV -> Pu                            *)
(* ============================================================================ *)

(* -------------------------------------------------------------------------- *)
(* 1) FBAI01_DI01  Senzori pritiska Pt (_0_0, _1.._6, _NS1, _NS2)            *)
(* Skaliranje raw AI -> bar. Parametri postavljeni u IO_Init.                 *)
(* -------------------------------------------------------------------------- *)
PG.Sens.Pt._0_0();  (* Pritisak komprimovanog vazduha, skalirani opseg -1 do 14 [bar] *)
PG.Sens.Pt._1();    (* Pritisak termalne vode na ulazu u podstanicu [bar] *)
PG.Sens.Pt._2();    (* Pritisak termalne vode posle streinera grubih filtera [bar] *)
PG.Sens.Pt._3();    (* Pritisak termalne vode posle velikog izmenjivaca [bar] *)
PG.Sens.Pt._4();    (* Pritisak termalne vode na ulazu u prihvatni tank [bar] *)
PG.Sens.Pt._5();    (* Pritisak na potisu transportnih pumpi [bar] *)
PG.Sens.Pt._6();    (* Dodatni transmiter pritiska [bar] *)
PG.Sens.Pt._NS1();  (* Pritisak na dnu prihvatnog tanka [bar] *)
PG.Sens.Pt._NS2();  (* Pritisak na vrhu prihvatnog tanka [bar] *)

(* -------------------------------------------------------------------------- *)
(* 2) FBAI01_DI01  Temperature TT_PG_01..TT_PG_11                         *)
(* Svi kanali su fizicki mapirani na X20AI4622b, X67AI1323 i X67AI1333b.    *)
(* -------------------------------------------------------------------------- *)
PG.Sens.Tt._1();  (* TT_PG_01 - ulaz u veliki razmenjivac PGRT01 [degC]. *)
PG.Sens.Tt._2();  (* TT_PG_02 - ulaz u prihvatni tank [degC]. *)
PG.Sens.Tt._3();  (* TT_PG_03 - temperatura u prihvatnom tanku [degC]. *)
PG.Sens.Tt._4();  (* TT_PG_04 - izlaz iz velikog razmenjivaca PGRT01 [degC]. *)
PG.Sens.Tt._5();  (* TT_PG_05 - ulaz u mali razmenjivac PGRT02 [degC]. *)
PG.Sens.Tt._6();  (* TT_PG_06 - izlaz iz malog razmenjivaca PGRT02 [degC]. *)
PG.Sens.Tt._7();  (* TT_PG_07 - drenazni vod za potvrdu zavrsetka preispiranja [degC]. *)
PG.Sens.Tt._8();  (* TT_PG_08 - ulaz tehnicke vode u direktni izmenjivac [degC]. *)
PG.Sens.Tt._9();  (* TT_PG_09 - izlaz tehnicke vode iz direktnog izmenjivaca [degC]. *)
PG.Sens.Tt._10(); (* TT_PG_10 - ulaz sanitarne vode u direktni izmenjivac [degC]. *)
PG.Sens.Tt._11(); (* TT_PG_11 - izlaz sanitarne vode iz direktnog izmenjivaca [degC]. *)

(* -------------------------------------------------------------------------- *)
(* 3) FBAI01_DI01  Merac protoka MP (_1)                                      *)
(* Skaliranje raw AI -> m3/h. TransmitterStatus DI aktivan (EnableStatusCheck).*)
(* -------------------------------------------------------------------------- *)
PG.Sens.MP._1();  (* Merac protoka na potisu tople termalne vode ka potrosacima [m3/h] *)

(* -------------------------------------------------------------------------- *)
(* 4) FB_DI  Nivo prekidaci LS (_1.._5)                                       *)
(* DI detekcija prisustva tecnosti u odzraci. DelayOn/Off=T#1s.               *)
(* -------------------------------------------------------------------------- *)
PG.Sens.LS._1();  (* Nizak nivo vode u prihvatnom tanku za rad pumpi *)
PG.Sens.LS._2();  (* Donji nivo u odzracnom cilindru na ulazu vode u podstanicu *)
PG.Sens.LS._3();  (* Gornji nivo u odzracnom cilindru na ulazu vode u podstanicu *)
PG.Sens.LS._4();  (* Donji nivo u odzracnom cilindru na ulazu vode u prihvatni tank *)
PG.Sens.LS._5();  (* Gornji nivo u odzracnom cilindru na ulazu vode u prihvatni tank *)

(* -------------------------------------------------------------------------- *)
(* 5) FB_DI  Prestrujni ventili OWF (_1, _2)                                  *)
(* DI povratni signal otvorenog polozaja. DelayOn/Off=T#500ms.                *)
(* -------------------------------------------------------------------------- *)
PG.Sens.OWF._1();  (* Zastitni prestrujni ventil od hidraulickog udara 1 *)
PG.Sens.OWF._2();  (* Zastitni prestrujni ventil od hidraulickog udara 2 *)

(* -------------------------------------------------------------------------- *)
(* 6) FB_V_EMV + FB_V_ON_OFF_FB  Automatski ventili AV (_1.._7)               *)
(* AV._1/2: bistabilni - CmdOpen i CmdClose mapirani u IoMap.                 *)
(* AV._3..AV._7: spring-return NC - samo Cmd mapiran u IoMap.                 *)
(* -------------------------------------------------------------------------- *)
PG.Act.AV._1();  (* Elektromotorni bistabilni leptir ventil DN125, OpenMaxTime=20s *)
PG.Act.AV._2();  (* Elektromotorni bistabilni leptir ventil DN125, OpenMaxTime=20s *)
PG.Act.AV._3();  (* Pneumatski NC spring-return leptir ventil DN125, OpenMaxTime=10s *)
PG.Act.AV._4();  (* Pneumatski NC spring-return leptir ventil DN125, OpenMaxTime=10s *)
PG.Act.AV._5();  (* Pneumatski NC spring-return leptir ventil DN125, OpenMaxTime=10s *)
PG.Act.AV._6();  (* Pneumatski NC spring-return leptir ventil DN125, OpenMaxTime=10s *)
PG.Act.AV._7();  (* Pneumatski NC spring-return leptir ventil DN125, OpenMaxTime=10s *)

(* -------------------------------------------------------------------------- *)
(* 7) FB_HV_2LS  Rucni leptir ventili RV (_19, _21.._27)                     *)
(* Monitoring 2 krajnja prekidaca, alarm pri timeout tranziciji.              *)
(* -------------------------------------------------------------------------- *)
PG.Act.RV._19();  (* Rucni ventil posle membranskog ventila PG_PV01 *)
PG.Act.RV._21();  (* Rucni ventil posle membranskog ventila PG_PV02 *)
PG.Act.RV._22();  (* Drenazni total ventil na dnu prihvatnog tanka *)
PG.Act.RV._23();  (* Ulaz u Pumpu PG_Pu01 *)
PG.Act.RV._24();  (* Ulaz u Pumpu PG_Pu02 *)
PG.Act.RV._25();  (* Bajpasni izlaz iz tanka ka instalaciji za izbacivanje gasa van kotlarnice *)
PG.Act.RV._26();  (* Ulaz u vakuum pumpu *)
PG.Act.RV._27();  (* Izlaz iz vakuum pumpe ka instalaciji za izbacivanje gasa van kotlarnice *)

(* -------------------------------------------------------------------------- *)
(* 9) FB_PvAiAo_Fast  Proporcionalni membranski ventili PV (_1.._5)           *)
(* AI_Raw povratni signal i AO_Raw komanda direktno mapirani u IoMap.         *)
(* -------------------------------------------------------------------------- *)

	PG.Act.PV._1(); (* Obrada granica, izbora Manual/Auto i AO komande PV._1. *)

	PG.Act.PV._2(); (* Obrada granica, izbora Manual/Auto i AO komande PV._2. *)

	PG.Act.PV._3(); (* Obrada granica, izbora Manual/Auto i AO komande PV._3. *)

	PG.Act.PV._4(); (* Obrada granica, izbora Manual/Auto i AO komande PV._4. *)

	PG.Act.PV._5(); (* Obrada granica, izbora Manual/Auto i AO komande PV._5. *)

(* -------------------------------------------------------------------------- *)
(* 10) vfdMain  Pumpe Pu (_1, _2)  DIO metod                                 *)
(* w_run_fwd/w_reset (DO) i w_freq (AO) mapirani u IoMap.                    *)
(* Trenutni clamp u kodu: Pu._1 = 10..100 Hz, Pu._2 = 10..50 Hz.             *)
(* addr_struct postavljen jednom u IO_Init tasku.                             *)
(* -------------------------------------------------------------------------- *)

	PG.Act.Pu.VFD_function._1();  (* Pumpa za snabdevanje potrosaca 01, Grundfoss CR45, METOD_DIO *)

	PG.Act.Pu.VFD_function._2();  (* Pumpa za snabdevanje potrosaca 02, Grundfoss CR45, METOD_DIO *)

END_PROGRAM
```

#### Exit.st
```iecst
PROGRAM _EXIT
	(* ======================================================================== *)
	(* IO_EXIT                                                                   *)
	(* Ovaj task trenutno nema posebnu gasnu proceduru.                          *)
	(* Svi FB-ovi i I/O signali prelaze u stanje definisano runtime-om i HW-om. *)
	(* ======================================================================== *)
END_PROGRAM
```

#### Init.st
```iecst
PROGRAM _INIT

(* ============================================================================ *)
(* IO_INIT  Inicijalizacija parametara za sve BR_Lib FB instance               *)
(* Objekat: PG  Podstanica grejanja 1, Kursumlijska Banja                     *)
(* IO veze: IoMap.iom  ovde su samo parametri i Enable politika.              *)
(* ============================================================================ *)

(* -------------------------------------------------------------------------- *)
(* 1) FBAI01_DI01  Senzori pritiska Pt (_1.._6)                               *)
(* X20AI4622 / X20AI4622a, 4-20mA, Cerabar PMP23. Opseg: -1...9 bara.        *)
(* ScaledMin=-1.0: zastitni offset jer 4mA odgovara 0 bara na terenu.        *)
(* -------------------------------------------------------------------------- *)
(* Pt._0_0: Pritisak komprimovanog vazduha [bar] *)
PG.Sens.Pt._0_0.AI_Input.Enable             := TRUE;      (* aktivira FB, pokrece skaliranje i statusnu logiku *)
PG.Sens.Pt._0_0.AI_Param.RawMin             := 0;         (* donja granica raw ADC opsega (0 = 4mA) *)
PG.Sens.Pt._0_0.AI_Param.RawMax             := 32767;     (* gornja granica raw ADC opsega (32767 = 20mA) *)
PG.Sens.Pt._0_0.AI_Param.ScaledMin          := -1.0;      (* donja fizicka vrednost opsega [bar] *)
PG.Sens.Pt._0_0.AI_Param.ScaledMax          := 15.0;      (* gornja fizicka vrednost opsega [bar] *)
PG.Sens.Pt._0_0.AI_Param.UnitOfMeasure      := 'bar';     (* jedinica za prikaz na HMI *)
PG.Sens.Pt._0_0.AI_Param.EnableStatusCheck  := FALSE;     (* bez TransmitterStatus DI - nije prikljucen *)

(* Pt._1: Pritisak termalne vode na ulazu u podstanicu [bar] *)
PG.Sens.Pt._1.AI_Input.Enable             := TRUE;      (* aktivira FB, pokrece skaliranje i statusnu logiku *)
PG.Sens.Pt._1.AI_Param.RawMin             := 0;         (* donja granica raw ADC opsega (0 = 4mA) *)
PG.Sens.Pt._1.AI_Param.RawMax             := 32767;     (* gornja granica raw ADC opsega (32767 = 20mA) *)
PG.Sens.Pt._1.AI_Param.ScaledMin          := -1.0;      (* 0-10 bar, offset -1: 4mA = 0 bar na terenu *)
PG.Sens.Pt._1.AI_Param.ScaledMax          := 9.0;       (* gornja fizicka vrednost opsega [bar] *)
PG.Sens.Pt._1.AI_Param.UnitOfMeasure      := 'bar';     (* jedinica za prikaz na HMI *)
PG.Sens.Pt._1.AI_Param.EnableStatusCheck  := FALSE;     (* bez TransmitterStatus DI - nije prikljucen *)

(* Pt._2: Pritisak termalne vode posle streinera grubih filtera [bar] *)
PG.Sens.Pt._2.AI_Input.Enable             := TRUE;      (* aktivira FB, pokrece skaliranje i statusnu logiku *)
PG.Sens.Pt._2.AI_Param.RawMin             := 0;         (* donja granica raw ADC opsega (0 = 4mA) *)
PG.Sens.Pt._2.AI_Param.RawMax             := 32767;     (* gornja granica raw ADC opsega (32767 = 20mA) *)
PG.Sens.Pt._2.AI_Param.ScaledMin          := -1.0;      (* 0-10 bar, offset -1: 4mA = 0 bar na terenu *)
PG.Sens.Pt._2.AI_Param.ScaledMax          := 9.0;       (* gornja fizicka vrednost opsega [bar] *)
PG.Sens.Pt._2.AI_Param.UnitOfMeasure      := 'bar';     (* jedinica za prikaz na HMI *)
PG.Sens.Pt._2.AI_Param.EnableStatusCheck  := FALSE;     (* bez TransmitterStatus DI - nije prikljucen *)

(* Pt._3: Pritisak termalne vode posle velikog izmenjivaca [bar] *)
PG.Sens.Pt._3.AI_Input.Enable             := TRUE;      (* aktivira FB, pokrece skaliranje i statusnu logiku *)
PG.Sens.Pt._3.AI_Param.RawMin             := 0;         (* donja granica raw ADC opsega (0 = 4mA) *)
PG.Sens.Pt._3.AI_Param.RawMax             := 32767;     (* gornja granica raw ADC opsega (32767 = 20mA) *)
PG.Sens.Pt._3.AI_Param.ScaledMin          := -1.0;      (* 0-10 bar, offset -1: 4mA = 0 bar na terenu *)
PG.Sens.Pt._3.AI_Param.ScaledMax          := 9.0;       (* gornja fizicka vrednost opsega [bar] *)
PG.Sens.Pt._3.AI_Param.UnitOfMeasure      := 'bar';     (* jedinica za prikaz na HMI *)
PG.Sens.Pt._3.AI_Param.EnableStatusCheck  := FALSE;     (* bez TransmitterStatus DI - nije prikljucen *)

(* Pt._4: Pritisak termalne vode na ulazu u prihvatni tank [bar] *)
PG.Sens.Pt._4.AI_Input.Enable             := TRUE;      (* aktivira FB, pokrece skaliranje i statusnu logiku *)
PG.Sens.Pt._4.AI_Param.RawMin             := 0;         (* donja granica raw ADC opsega (0 = 4mA) *)
PG.Sens.Pt._4.AI_Param.RawMax             := 32767;     (* gornja granica raw ADC opsega (32767 = 20mA) *)
PG.Sens.Pt._4.AI_Param.ScaledMin          := -1.0;      (* 0-10 bar, offset -1: 4mA = 0 bar na terenu *)
PG.Sens.Pt._4.AI_Param.ScaledMax          := 9.0;       (* gornja fizicka vrednost opsega [bar] *)
PG.Sens.Pt._4.AI_Param.UnitOfMeasure      := 'bar';     (* jedinica za prikaz na HMI *)
PG.Sens.Pt._4.AI_Param.EnableStatusCheck  := FALSE;     (* bez TransmitterStatus DI - nije prikljucen *)

(* Pt._5: Pritisak na potisu transportnih pumpi [bar] *)
PG.Sens.Pt._5.AI_Input.Enable             := TRUE;      (* aktivira FB, pokrece skaliranje i statusnu logiku *)
PG.Sens.Pt._5.AI_Param.RawMin             := 0;         (* donja granica raw ADC opsega (0 = 4mA) *)
PG.Sens.Pt._5.AI_Param.RawMax             := 32767;     (* gornja granica raw ADC opsega (32767 = 20mA) *)
PG.Sens.Pt._5.AI_Param.ScaledMin          := -1.0;      (* 0-10 bar, offset -1: 4mA = 0 bar na terenu *)
PG.Sens.Pt._5.AI_Param.ScaledMax          := 9.0;       (* gornja fizicka vrednost opsega [bar] *)
PG.Sens.Pt._5.AI_Param.UnitOfMeasure      := 'bar';     (* jedinica za prikaz na HMI *)
PG.Sens.Pt._5.AI_Param.EnableStatusCheck  := FALSE;     (* bez TransmitterStatus DI - nije prikljucen *)

(* Pt._6: Dodatni transmiter pritiska [bar] *)
PG.Sens.Pt._6.AI_Input.Enable             := TRUE;      (* aktivira FB, pokrece skaliranje i statusnu logiku *)
PG.Sens.Pt._6.AI_Param.RawMin             := 0;         (* donja granica raw ADC opsega (0 = 4mA) *)
PG.Sens.Pt._6.AI_Param.RawMax             := 32767;     (* gornja granica raw ADC opsega (32767 = 20mA) *)
PG.Sens.Pt._6.AI_Param.ScaledMin          := -1.0;      (* 0-10 bar, offset -1: 4mA = 0 bar na terenu *)
PG.Sens.Pt._6.AI_Param.ScaledMax          := 9.0;       (* gornja fizicka vrednost opsega [bar] *)
PG.Sens.Pt._6.AI_Param.UnitOfMeasure      := 'bar';     (* jedinica za prikaz na HMI *)
PG.Sens.Pt._6.AI_Param.EnableStatusCheck  := FALSE;     (* bez TransmitterStatus DI - nije prikljucen *)

(* -------------------------------------------------------------------------- *)
(* 2) FBAI01_DI01  Senzori niskog pritiska Pt (_NS1, _NS2) za merenje nivoa  *)
(* X20AI4622a, 4-20mA, Cerabar PMP23. Opseg: -0.1...0.3 bar (PTNS).          *)
(* -------------------------------------------------------------------------- *)
(* Pt._NS1: Pritisak na dnu prihvatnog tanka [bar] *)
PG.Sens.Pt._NS1.AI_Input.Enable             := TRUE;    (* aktivira FB, pokrece skaliranje i statusnu logiku *)
PG.Sens.Pt._NS1.AI_Param.RawMin             := 0;       (* donja granica raw ADC opsega (0 = 4mA) *)
PG.Sens.Pt._NS1.AI_Param.RawMax             := 32767;   (* gornja granica raw ADC opsega (32767 = 20mA) *)
PG.Sens.Pt._NS1.AI_Param.ScaledMin          := -0.1;  (* donja fizicka vrednost opsega [bar] *)
PG.Sens.Pt._NS1.AI_Param.ScaledMax          := 0.3;   (* gornja fizicka vrednost opsega [bar] *)
PG.Sens.Pt._NS1.AI_Param.UnitOfMeasure      := 'bar';  (* jedinica za prikaz na HMI *)
PG.Sens.Pt._NS1.AI_Param.EnableStatusCheck  := FALSE;   (* bez TransmitterStatus DI - nije prikljucen *)

(* Pt._NS2: Pritisak na vrhu prihvatnog tanka [bar] *)
PG.Sens.Pt._NS2.AI_Input.Enable             := TRUE;    (* aktivira FB, pokrece skaliranje i statusnu logiku *)
PG.Sens.Pt._NS2.AI_Param.RawMin             := 0;       (* donja granica raw ADC opsega (0 = 4mA) *)
PG.Sens.Pt._NS2.AI_Param.RawMax             := 32767;   (* gornja granica raw ADC opsega (32767 = 20mA) *)
PG.Sens.Pt._NS2.AI_Param.ScaledMin          := -0.1;  (* donja fizicka vrednost opsega [bar] *)
PG.Sens.Pt._NS2.AI_Param.ScaledMax          := 0.3;   (* gornja fizicka vrednost opsega [bar] *)
PG.Sens.Pt._NS2.AI_Param.UnitOfMeasure      := 'bar';  (* jedinica za prikaz na HMI *)
PG.Sens.Pt._NS2.AI_Param.EnableStatusCheck  := FALSE;   (* bez TransmitterStatus DI - nije prikljucen *)

(* -------------------------------------------------------------------------- *)
(* 3) FBAI01_DI01  Temperature TT_PG_01..TT_PG_07                             *)
(* TT_PG_01..03 su mapirani na X20AI4622b; TT_PG_04..07 cekaju AI mapiranje.   *)
(* Easytemp TMR35, 4-20mA. Opseg: 0-120 degC.                                  *)
(* -------------------------------------------------------------------------- *)
(* Tt._1 / TT_PG_01: Ulaz u veliki razmenjivac PGRT01 [degC]. *)
PG.Sens.Tt._1.AI_Input.Enable             := TRUE;      (* Aktivira obradu mapiranog AI signala. *)
PG.Sens.Tt._1.AI_Param.RawMin             := 0;         (* 4 mA. *)
PG.Sens.Tt._1.AI_Param.RawMax             := 32767;     (* 20 mA. *)
PG.Sens.Tt._1.AI_Param.ScaledMin          := 0.0;       (* Donja granica [degC]. *)
PG.Sens.Tt._1.AI_Param.ScaledMax          := 120.0;     (* Gornja granica [degC]. *)
PG.Sens.Tt._1.AI_Param.UnitOfMeasure      := 'degC';    (* HMI jedinica. *)
PG.Sens.Tt._1.AI_Param.EnableStatusCheck  := FALSE;     (* Nema statusnog DI signala. *)

(* Tt._2 / TT_PG_02: Temperatura na ulazu u prihvatni tank [degC]. *)
PG.Sens.Tt._2.AI_Input.Enable             := TRUE;      (* Aktivira obradu mapiranog AI signala. *)
PG.Sens.Tt._2.AI_Param.RawMin             := 0;         (* 4 mA. *)
PG.Sens.Tt._2.AI_Param.RawMax             := 32767;     (* 20 mA. *)
PG.Sens.Tt._2.AI_Param.ScaledMin          := 0.0;       (* Donja granica [degC]. *)
PG.Sens.Tt._2.AI_Param.ScaledMax          := 120.0;     (* Gornja granica [degC]. *)
PG.Sens.Tt._2.AI_Param.UnitOfMeasure      := 'degC';    (* HMI jedinica. *)
PG.Sens.Tt._2.AI_Param.EnableStatusCheck  := FALSE;     (* Nema statusnog DI signala. *)

(* Tt._3 / TT_PG_03: Temperatura u prihvatnom tanku [degC]. *)
PG.Sens.Tt._3.AI_Input.Enable             := TRUE;      (* Aktivira obradu mapiranog AI signala. *)
PG.Sens.Tt._3.AI_Param.RawMin             := 0;         (* 4 mA. *)
PG.Sens.Tt._3.AI_Param.RawMax             := 32767;     (* 20 mA. *)
PG.Sens.Tt._3.AI_Param.ScaledMin          := 0.0;       (* Donja granica [degC]. *)
PG.Sens.Tt._3.AI_Param.ScaledMax          := 120.0;     (* Gornja granica [degC]. *)
PG.Sens.Tt._3.AI_Param.UnitOfMeasure      := 'degC';    (* HMI jedinica. *)
PG.Sens.Tt._3.AI_Param.EnableStatusCheck  := FALSE;     (* Nema statusnog DI signala. *)

(* Tt._4 / TT_PG_04: Izlaz iz velikog razmenjivaca PGRT01 [degC]. *)
PG.Sens.Tt._4.AI_Input.Enable             := TRUE;      (* Aktivira obradu mapiranog AI signala. *)
PG.Sens.Tt._4.AI_Param.RawMin             := 0;         (* 4 mA. *)
PG.Sens.Tt._4.AI_Param.RawMax             := 32767;     (* 20 mA. *)
PG.Sens.Tt._4.AI_Param.ScaledMin          := 0.0;       (* Donja granica [degC]. *)
PG.Sens.Tt._4.AI_Param.ScaledMax          := 120.0;     (* Gornja granica [degC]. *)
PG.Sens.Tt._4.AI_Param.UnitOfMeasure      := 'degC';    (* HMI jedinica. *)
PG.Sens.Tt._4.AI_Param.EnableStatusCheck  := FALSE;     (* Nema statusnog DI signala. *)

(* Tt._5 / TT_PG_05: Ulaz u mali razmenjivac PGRT02 [degC]. *)
PG.Sens.Tt._5.AI_Input.Enable             := TRUE;      (* Aktivira obradu mapiranog AI signala. *)
PG.Sens.Tt._5.AI_Param.RawMin             := 0;         (* 4 mA. *)
PG.Sens.Tt._5.AI_Param.RawMax             := 32767;     (* 20 mA. *)
PG.Sens.Tt._5.AI_Param.ScaledMin          := 0.0;       (* Donja granica [degC]. *)
PG.Sens.Tt._5.AI_Param.ScaledMax          := 120.0;     (* Gornja granica [degC]. *)
PG.Sens.Tt._5.AI_Param.UnitOfMeasure      := 'degC';    (* HMI jedinica. *)
PG.Sens.Tt._5.AI_Param.EnableStatusCheck  := FALSE;     (* Nema statusnog DI signala. *)

(* Tt._6 / TT_PG_06: Izlaz iz malog razmenjivaca PGRT02 [degC]. *)
PG.Sens.Tt._6.AI_Input.Enable             := TRUE;      (* Aktivira obradu mapiranog AI signala. *)
PG.Sens.Tt._6.AI_Param.RawMin             := 0;         (* 4 mA. *)
PG.Sens.Tt._6.AI_Param.RawMax             := 32767;     (* 20 mA. *)
PG.Sens.Tt._6.AI_Param.ScaledMin          := 0.0;       (* Donja granica [degC]. *)
PG.Sens.Tt._6.AI_Param.ScaledMax          := 120.0;     (* Gornja granica [degC]. *)
PG.Sens.Tt._6.AI_Param.UnitOfMeasure      := 'degC';    (* HMI jedinica. *)
PG.Sens.Tt._6.AI_Param.EnableStatusCheck  := FALSE;     (* Nema statusnog DI signala. *)

(* Tt._7 / TT_PG_07: Drenazni vod za potvrdu zavrsetka preispiranja [degC]. *)
PG.Sens.Tt._7.AI_Input.Enable             := TRUE;      (* Aktivira obradu mapiranog AI signala. *)
PG.Sens.Tt._7.AI_Param.RawMin             := 0;         (* 4 mA. *)
PG.Sens.Tt._7.AI_Param.RawMax             := 32767;     (* 20 mA. *)
PG.Sens.Tt._7.AI_Param.ScaledMin          := 0.0;       (* Donja granica [degC]. *)
PG.Sens.Tt._7.AI_Param.ScaledMax          := 120.0;     (* Gornja granica [degC]. *)
PG.Sens.Tt._7.AI_Param.UnitOfMeasure      := 'degC';    (* HMI jedinica. *)
PG.Sens.Tt._7.AI_Param.EnableStatusCheck  := FALSE;     (* Nema statusnog DI signala. *)

(* -------------------------------------------------------------------------- *)
(* 3.1) FBAI01_DI01  Temperature TT_PG_08..TT_PG_11                        *)
(* Tehnicka i sanitarna voda kroz direktni izmenjivac, 0..120 degC.          *)
(* -------------------------------------------------------------------------- *)
(* Tt._8 / TT_PG_08: ulaz tehnicke vode u direktni izmenjivac [degC]. *)
PG.Sens.Tt._8.AI_Input.Enable             := TRUE;      (* Aktivira obradu mapiranog AI signala. *)
PG.Sens.Tt._8.AI_Param.RawMin             := 0;         (* 4 mA. *)
PG.Sens.Tt._8.AI_Param.RawMax             := 32767;     (* 20 mA. *)
PG.Sens.Tt._8.AI_Param.ScaledMin          := 0.0;       (* Donja granica [degC]. *)
PG.Sens.Tt._8.AI_Param.ScaledMax          := 120.0;     (* Gornja granica [degC]. *)
PG.Sens.Tt._8.AI_Param.UnitOfMeasure      := 'degC';    (* HMI jedinica. *)
PG.Sens.Tt._8.AI_Param.EnableStatusCheck  := FALSE;     (* Nema statusnog DI signala. *)

(* Tt._9 / TT_PG_09: izlaz tehnicke vode iz direktnog izmenjivaca [degC]. *)
PG.Sens.Tt._9.AI_Input.Enable             := TRUE;      (* Aktivira obradu mapiranog AI signala. *)
PG.Sens.Tt._9.AI_Param.RawMin             := 0;         (* 4 mA. *)
PG.Sens.Tt._9.AI_Param.RawMax             := 32767;     (* 20 mA. *)
PG.Sens.Tt._9.AI_Param.ScaledMin          := 0.0;       (* Donja granica [degC]. *)
PG.Sens.Tt._9.AI_Param.ScaledMax          := 120.0;     (* Gornja granica [degC]. *)
PG.Sens.Tt._9.AI_Param.UnitOfMeasure      := 'degC';    (* HMI jedinica. *)
PG.Sens.Tt._9.AI_Param.EnableStatusCheck  := FALSE;     (* Nema statusnog DI signala. *)

(* Tt._10 / TT_PG_10: ulaz sanitarne vode u direktni izmenjivac [degC]. *)
PG.Sens.Tt._10.AI_Input.Enable            := TRUE;      (* Aktivira obradu mapiranog AI signala. *)
PG.Sens.Tt._10.AI_Param.RawMin            := 0;         (* 4 mA. *)
PG.Sens.Tt._10.AI_Param.RawMax            := 32767;     (* 20 mA. *)
PG.Sens.Tt._10.AI_Param.ScaledMin         := 0.0;       (* Donja granica [degC]. *)
PG.Sens.Tt._10.AI_Param.ScaledMax         := 120.0;     (* Gornja granica [degC]. *)
PG.Sens.Tt._10.AI_Param.UnitOfMeasure     := 'degC';    (* HMI jedinica. *)
PG.Sens.Tt._10.AI_Param.EnableStatusCheck := FALSE;     (* Nema statusnog DI signala. *)

(* Tt._11 / TT_PG_11: izlaz sanitarne vode iz direktnog izmenjivaca [degC]. *)
PG.Sens.Tt._11.AI_Input.Enable            := TRUE;      (* Aktivira obradu mapiranog AI signala. *)
PG.Sens.Tt._11.AI_Param.RawMin            := 0;         (* 4 mA. *)
PG.Sens.Tt._11.AI_Param.RawMax            := 32767;     (* 20 mA. *)
PG.Sens.Tt._11.AI_Param.ScaledMin         := 0.0;       (* Donja granica [degC]. *)
PG.Sens.Tt._11.AI_Param.ScaledMax         := 120.0;     (* Gornja granica [degC]. *)
PG.Sens.Tt._11.AI_Param.UnitOfMeasure     := 'degC';    (* HMI jedinica. *)
PG.Sens.Tt._11.AI_Param.EnableStatusCheck := FALSE;     (* Nema statusnog DI signala. *)

(* -------------------------------------------------------------------------- *)
(* 4) FBAI01_DI01  Merac protoka MP (_1)                                      *)
(* X20AI4622c AI01, 4-20mA, Promag H10 DN065. Opseg: 0-10 l/s.                *)
(* EnableStatusCheck=TRUE: TransmitterStatus DI mapiran u IoMap.              *)
(* -------------------------------------------------------------------------- *)
(* MP._1: Merac protoka na potisu tople termalne vode ka potrosacima [m3/h]  *)
PG.Sens.MP._1.AI_Input.Enable             := TRUE;      (* aktivira FB, pokrece skaliranje i statusnu logiku *)
PG.Sens.MP._1.AI_Param.RawMin             := 0;         (* donja granica raw ADC opsega (0 = 4mA) *)
PG.Sens.MP._1.AI_Param.RawMax             := 32767;     (* gornja granica raw ADC opsega (32767 = 20mA) *)
PG.Sens.MP._1.AI_Param.ScaledMin          := 0.0;       (* min protok [m3/h], 0 l/s *)
PG.Sens.MP._1.AI_Param.ScaledMax          := 20.0;      (* max protok [m3/h], 20 l/s *)
PG.Sens.MP._1.AI_Param.UnitOfMeasure      := 'l/s';    (* jedinica za prikaz na HMI *)
PG.Sens.MP._1.AI_Param.EnableStatusCheck  := TRUE;      (* Promag H10 status DI aktivan, mapiran u IoMap *)

(* -------------------------------------------------------------------------- *)
(* 5) FB_DI  Nivo prekidaci LS (_1.._5)                                       *)
(* Liquipoint FTW23, Tri clamp DN040: detekcija prisustva tecnosti u odzraci. *)
(* DelayOn/Off=T#1s za filtriranje kratkih tranzijenta.                       *)
(* -------------------------------------------------------------------------- *)
(* LS._1: Nizak nivo vode u prihvatnom tanku za rad pumpi *)
PG.Sens.LS._1.DI_Input.Enable          := TRUE;         (* aktivira FB pracenja DI signala *)
PG.Sens.LS._1.DI_Param.UseStatusInput  := FALSE;        (* nema poseban DI za status uredaja *)
PG.Sens.LS._1.DI_Param.InvertSignal    := FALSE;        (* signal se NE invertuje *)
PG.Sens.LS._1.DI_Param.DelayOn         := T#1s;         (* kasnjenje aktivacije - filtriranje tranzijenta *)
PG.Sens.LS._1.DI_Param.DelayOff        := T#1s;         (* kasnjenje deaktivacije - filtriranje tranzijenta *)
PG.Sens.LS._1.DI_Param.TextTrue        := 'Tecnost prisutna';  (* tekst za HMI kada je DI aktivan *)
PG.Sens.LS._1.DI_Param.TextFalse       := 'Tecnost odsutna';   (* tekst za HMI kada je DI neaktivan *)
PG.Sens.LS._1.DI_Param.TextAlarm       := 'LS alarm';   (* tekst alarma za HMI i logovanje *)
PG.Sens.LS._1.DI_Param.TextFault       := 'LS fault';   (* tekst kvara za HMI i logovanje *)

(* LS._2: Donji nivo u odzracnom cilindru na ulazu vode u podstanicu *)
PG.Sens.LS._2.DI_Input.Enable          := TRUE;         (* aktivira FB pracenja DI signala *)
PG.Sens.LS._2.DI_Param.UseStatusInput  := FALSE;        (* nema poseban DI za status uredaja *)
PG.Sens.LS._2.DI_Param.InvertSignal    := FALSE;        (* signal se NE invertuje *)
PG.Sens.LS._2.DI_Param.DelayOn         := T#1s;         (* kasnjenje aktivacije - filtriranje tranzijenta *)
PG.Sens.LS._2.DI_Param.DelayOff        := T#1s;         (* kasnjenje deaktivacije - filtriranje tranzijenta *)
PG.Sens.LS._2.DI_Param.TextTrue        := 'Tecnost prisutna';  (* tekst za HMI kada je DI aktivan *)
PG.Sens.LS._2.DI_Param.TextFalse       := 'Tecnost odsutna';   (* tekst za HMI kada je DI neaktivan *)
PG.Sens.LS._2.DI_Param.TextAlarm       := 'LS alarm';   (* tekst alarma za HMI i logovanje *)
PG.Sens.LS._2.DI_Param.TextFault       := 'LS fault';   (* tekst kvara za HMI i logovanje *)

(* LS._3: Gornji nivo u odzracnom cilindru na ulazu vode u podstanicu *)
PG.Sens.LS._3.DI_Input.Enable          := TRUE;         (* aktivira FB pracenja DI signala *)
PG.Sens.LS._3.DI_Param.UseStatusInput  := FALSE;        (* nema poseban DI za status uredaja *)
PG.Sens.LS._3.DI_Param.InvertSignal    := FALSE;        (* signal se NE invertuje *)
PG.Sens.LS._3.DI_Param.DelayOn         := T#1s;         (* kasnjenje aktivacije - filtriranje tranzijenta *)
PG.Sens.LS._3.DI_Param.DelayOff        := T#1s;         (* kasnjenje deaktivacije - filtriranje tranzijenta *)
PG.Sens.LS._3.DI_Param.TextTrue        := 'Tecnost prisutna';  (* tekst za HMI kada je DI aktivan *)
PG.Sens.LS._3.DI_Param.TextFalse       := 'Tecnost odsutna';   (* tekst za HMI kada je DI neaktivan *)
PG.Sens.LS._3.DI_Param.TextAlarm       := 'LS alarm';   (* tekst alarma za HMI i logovanje *)
PG.Sens.LS._3.DI_Param.TextFault       := 'LS fault';   (* tekst kvara za HMI i logovanje *)

(* LS._4: Donji nivo u odzracnom cilindru na ulazu vode u prihvatni tank *)
PG.Sens.LS._4.DI_Input.Enable          := TRUE;         (* aktivira FB pracenja DI signala *)
PG.Sens.LS._4.DI_Param.UseStatusInput  := FALSE;        (* nema poseban DI za status uredaja *)
PG.Sens.LS._4.DI_Param.InvertSignal    := FALSE;        (* signal se NE invertuje *)
PG.Sens.LS._4.DI_Param.DelayOn         := T#1s;         (* kasnjenje aktivacije - filtriranje tranzijenta *)
PG.Sens.LS._4.DI_Param.DelayOff        := T#1s;         (* kasnjenje deaktivacije - filtriranje tranzijenta *)
PG.Sens.LS._4.DI_Param.TextTrue        := 'Tecnost prisutna';  (* tekst za HMI kada je DI aktivan *)
PG.Sens.LS._4.DI_Param.TextFalse       := 'Tecnost odsutna';   (* tekst za HMI kada je DI neaktivan *)
PG.Sens.LS._4.DI_Param.TextAlarm       := 'LS alarm';   (* tekst alarma za HMI i logovanje *)
PG.Sens.LS._4.DI_Param.TextFault       := 'LS fault';   (* tekst kvara za HMI i logovanje *)

(* LS._5: Gornji nivo u odzracnom cilindru na ulazu vode u prihvatni tank *)
PG.Sens.LS._5.DI_Input.Enable          := TRUE;         (* aktivira FB pracenja DI signala *)
PG.Sens.LS._5.DI_Param.UseStatusInput  := FALSE;        (* nema poseban DI za status uredaja *)
PG.Sens.LS._5.DI_Param.InvertSignal    := FALSE;        (* signal se NE invertuje *)
PG.Sens.LS._5.DI_Param.DelayOn         := T#1s;         (* kasnjenje aktivacije - filtriranje tranzijenta *)
PG.Sens.LS._5.DI_Param.DelayOff        := T#1s;         (* kasnjenje deaktivacije - filtriranje tranzijenta *)
PG.Sens.LS._5.DI_Param.TextTrue        := 'Tecnost prisutna';  (* tekst za HMI kada je DI aktivan *)
PG.Sens.LS._5.DI_Param.TextFalse       := 'Tecnost odsutna';   (* tekst za HMI kada je DI neaktivan *)
PG.Sens.LS._5.DI_Param.TextAlarm       := 'LS alarm';   (* tekst alarma za HMI i logovanje *)
PG.Sens.LS._5.DI_Param.TextFault       := 'LS fault';   (* tekst kvara za HMI i logovanje *)

(* -------------------------------------------------------------------------- *)
(* 6) FB_DI  Prestrujni ventili OWF (_1, _2)                                  *)
(* NIOB FLUID 5371 DN050, povratni signal otvorenog polozaja 3-5 bara.        *)
(* DelayOn/Off=T#500ms za filtriranje kratkih tranzijenta pri promeni pritiska.*)
(* -------------------------------------------------------------------------- *)
(* OWF._1: Zastitni prestrujni ventil od hidraulickog udara 1 *)
PG.Sens.OWF._1.DI_Input.Enable          := TRUE;        (* aktivira FB pracenja DI signala *)
PG.Sens.OWF._1.DI_Param.UseStatusInput  := FALSE;       (* nema poseban DI za status uredaja *)
PG.Sens.OWF._1.DI_Param.InvertSignal    := FALSE;       (* signal se NE invertuje *)
PG.Sens.OWF._1.DI_Param.DelayOn         := T#500ms;     (* kasnjenje aktivacije - filtriranje pri promeni pritiska *)
PG.Sens.OWF._1.DI_Param.DelayOff        := T#500ms;     (* kasnjenje deaktivacije - filtriranje pri promeni pritiska *)
PG.Sens.OWF._1.DI_Param.TextTrue        := 'OWF otvoren';   (* tekst za HMI kada je ventil otvoren *)
PG.Sens.OWF._1.DI_Param.TextFalse       := 'OWF zatvoren';  (* tekst za HMI kada je ventil zatvoren *)
PG.Sens.OWF._1.DI_Param.TextAlarm       := 'OWF alarm';     (* tekst alarma za HMI i logovanje *)
PG.Sens.OWF._1.DI_Param.TextFault       := 'OWF fault';     (* tekst kvara za HMI i logovanje *)

(* OWF._2: Zastitni prestrujni ventil od hidraulickog udara 2 *)
PG.Sens.OWF._2.DI_Input.Enable          := TRUE;        (* aktivira FB pracenja DI signala *)
PG.Sens.OWF._2.DI_Param.UseStatusInput  := FALSE;       (* nema poseban DI za status uredaja *)
PG.Sens.OWF._2.DI_Param.InvertSignal    := FALSE;       (* signal se NE invertuje *)
PG.Sens.OWF._2.DI_Param.DelayOn         := T#500ms;     (* kasnjenje aktivacije - filtriranje pri promeni pritiska *)
PG.Sens.OWF._2.DI_Param.DelayOff        := T#500ms;     (* kasnjenje deaktivacije - filtriranje pri promeni pritiska *)
PG.Sens.OWF._2.DI_Param.TextTrue        := 'OWF otvoren';   (* tekst za HMI kada je ventil otvoren *)
PG.Sens.OWF._2.DI_Param.TextFalse       := 'OWF zatvoren';  (* tekst za HMI kada je ventil zatvoren *)
PG.Sens.OWF._2.DI_Param.TextAlarm       := 'OWF alarm';     (* tekst alarma za HMI i logovanje *)
PG.Sens.OWF._2.DI_Param.TextFault       := 'OWF fault';     (* tekst kvara za HMI i logovanje *)

(* -------------------------------------------------------------------------- *)
(* 7) FB_V_EMV + FB_V_ON_OFF_FB  Automatski ventili AV (_1.._7)               *)
(* AV._1, _2: End Armaturen DN125, elektromotorni bistabilni, CmdOpen+CmdClose*)
(* AV._3.._7: End Armaturen DN125, pneumatski NC spring-return, samo Cmd.     *)
(* OpenMaxTime: bistabilni=20s, spring-return=10s.                             *)
(* AV._1/_2 koriste PositionConfirmTime; AV._3.._7 koriste StableFbDelay.     *)
(* -------------------------------------------------------------------------- *)
(* AV._1: Elektromotorni leptir ventil DN125 bistabilan  razmenjivac toplote *)
PG.Act.AV._1.V_Input.Enable            := FALSE;         (* aktivira FB upravljanja ventilom *)
PG.Act.AV._1.V_Input.ForceCmd      	   := FALSE;         (* komanda ide na izlaz bez obzira na stanje / alarm *)
PG.Act.AV._1.V_Param.LampOpenExists    := TRUE;         (* pomocni DI signal LampOpen je dostupan i koristi se u logici FB-a *)
PG.Act.AV._1.V_Param.LampCloseExists   := TRUE;         (* pomocni DI signal LampClose je dostupan i koristi se u logici FB-a *)
PG.Act.AV._1.V_Param.OpenFbExists      := TRUE;         (* postoji DI povratni signal za otvoreni polozaj *)
PG.Act.AV._1.V_Param.CloseFbExists     := TRUE;         (* postoji DI povratni signal za zatvoreni polozaj *)
PG.Act.AV._1.V_Param.OverTorqueExists  := TRUE;         (* postoji DI signal preopterecenja za AV._1 *)
PG.Act.AV._1.V_Param.OpenMaxTime       := T#20s;        (* timeout - alarm ako FB otvoren ne stigne za 20s *)
PG.Act.AV._1.V_Param.CloseMaxTime      := T#20s;        (* timeout - alarm ako FB zatvoren ne stigne za 20s *)
PG.Act.AV._1.V_Param.EndLimitFilterTime := T#50ms;      (* filtriranje LampOpen/LampClose signala pre evaluacije stanja *)
PG.Act.AV._1.V_Param.PositionFbFilterTime := T#100ms;   (* filtriranje OpenFb/CloseFb signala pre potvrde pozicije *)
PG.Act.AV._1.V_Param.OverTorqueFilterTime := T#20ms;    (* filtriranje preopterecenja pre formiranja fault uslova *)
PG.Act.AV._1.V_Param.PositionConfirmTime := T#2s;       (* vreme cekanja trajnog feedback-a nakon krajnjeg polozaja *)

(* AV._2: Elektromotorni leptir ventil DN125 bistabilan  razmenjivac toplote *)
PG.Act.AV._2.V_Input.Enable            := FALSE;         (* aktivira FB upravljanja ventilom *)
PG.Act.AV._2.V_Input.ForceCmd      	   := FALSE;         (* komanda ide na izlaz bez obzira na stanje / alarm *)
PG.Act.AV._2.V_Param.LampOpenExists    := TRUE;         (* pomocni DI signal LampOpen je dostupan i koristi se u logici FB-a *)
PG.Act.AV._2.V_Param.LampCloseExists   := TRUE;         (* pomocni DI signal LampClose je dostupan i koristi se u logici FB-a *)
PG.Act.AV._2.V_Param.OpenFbExists      := TRUE;         (* postoji DI povratni signal za otvoreni polozaj *)
PG.Act.AV._2.V_Param.CloseFbExists     := TRUE;         (* postoji DI povratni signal za zatvoreni polozaj *)
PG.Act.AV._2.V_Param.OverTorqueExists  := FALSE;        (* AV._2 nema fizicki DI signal preopterecenja *)
PG.Act.AV._2.V_Param.OpenMaxTime       := T#20s;        (* timeout - alarm ako FB otvoren ne stigne za 20s *)
PG.Act.AV._2.V_Param.CloseMaxTime      := T#20s;        (* timeout - alarm ako FB zatvoren ne stigne za 20s *)
PG.Act.AV._2.V_Param.EndLimitFilterTime := T#50ms;      (* filtriranje LampOpen/LampClose signala pre evaluacije stanja *)
PG.Act.AV._2.V_Param.PositionFbFilterTime := T#100ms;   (* filtriranje OpenFb/CloseFb signala pre potvrde pozicije *)
PG.Act.AV._2.V_Param.PositionConfirmTime := T#2s;       (* vreme cekanja trajnog feedback-a nakon krajnjeg polozaja *)

(* AV._3: Pneumatski NC leptir ventil DN125 spring-return  prihvatni tank 1 *)
PG.Act.AV._3.V_Input.Enable            := TRUE;         (* aktivira FB upravljanja ventilom *)
PG.Act.AV._3.V_Input.ForceCmd      	   := TRUE;         (* komanda ide na izlaz bez obzira na stanje / alarm *)
PG.Act.AV._3.V_Param.FbOpenExists      := TRUE;         (* postoji DI povratni signal za otvoreni polozaj *)
PG.Act.AV._3.V_Param.FbCloseExists     := TRUE;         (* postoji DI povratni signal za zatvoreni polozaj *)
PG.Act.AV._3.V_Param.OpenMinTime       := T#0s;         (* min vreme drzanja komande otvori pre provere FB *)
PG.Act.AV._3.V_Param.OpenMaxTime       := T#10s;        (* timeout - spring-return brzi od elektromotornog *)
PG.Act.AV._3.V_Param.CloseMinTime      := T#0s;         (* min vreme drzanja komande zatvori pre provere FB *)
PG.Act.AV._3.V_Param.CloseMaxTime      := T#10s;        (* timeout - spring-return brzi od elektromotornog *)
PG.Act.AV._3.V_Param.StableFbDelay     := T#2s;         (* vreme stabilizacije FB signala pre potvrde polozaja *)

(* AV._4: Pneumatski NC leptir ventil DN125 spring-return  prihvatni tank 2 *)
PG.Act.AV._4.V_Input.Enable            := TRUE;         (* aktivira FB upravljanja ventilom *)
PG.Act.AV._4.V_Input.ForceCmd      	   := TRUE;         (* komanda ide na izlaz bez obzira na stanje / alarm *)
PG.Act.AV._4.V_Param.FbOpenExists      := TRUE;         (* postoji DI povratni signal za otvoreni polozaj *)
PG.Act.AV._4.V_Param.FbCloseExists     := TRUE;         (* postoji DI povratni signal za zatvoreni polozaj *)
PG.Act.AV._4.V_Param.OpenMinTime       := T#0s;         (* min vreme drzanja komande otvori pre provere FB *)
PG.Act.AV._4.V_Param.OpenMaxTime       := T#10s;        (* timeout - spring-return brzi od elektromotornog *)
PG.Act.AV._4.V_Param.CloseMinTime      := T#0s;         (* min vreme drzanja komande zatvori pre provere FB *)
PG.Act.AV._4.V_Param.CloseMaxTime      := T#10s;        (* timeout - spring-return brzi od elektromotornog *)
PG.Act.AV._4.V_Param.StableFbDelay     := T#2s;         (* vreme stabilizacije FB signala pre potvrde polozaja *)

(* AV._5: Pneumatski NC leptir ventil DN125 spring-return *)
PG.Act.AV._5.V_Input.Enable            := TRUE;         (* aktivira FB upravljanja ventilom *)
PG.Act.AV._5.V_Input.ForceCmd      	   := TRUE;         (* komanda ide na izlaz bez obzira na stanje / alarm *)
PG.Act.AV._5.V_Param.FbOpenExists      := TRUE;         (* postoji DI povratni signal za otvoreni polozaj *)
PG.Act.AV._5.V_Param.FbCloseExists     := TRUE;         (* postoji DI povratni signal za zatvoreni polozaj *)
PG.Act.AV._5.V_Param.OpenMinTime       := T#0s;         (* min vreme drzanja komande otvori pre provere FB *)
PG.Act.AV._5.V_Param.OpenMaxTime       := T#10s;        (* timeout - spring-return brzi od elektromotornog *)
PG.Act.AV._5.V_Param.CloseMinTime      := T#0s;         (* min vreme drzanja komande zatvori pre provere FB *)
PG.Act.AV._5.V_Param.CloseMaxTime      := T#10s;        (* timeout - spring-return brzi od elektromotornog *)
PG.Act.AV._5.V_Param.StableFbDelay     := T#2s;         (* vreme stabilizacije FB signala pre potvrde polozaja *)

(* AV._6: Pneumatski NC leptir ventil DN125 spring-return *)
PG.Act.AV._6.V_Input.Enable            := TRUE;         (* aktivira FB upravljanja ventilom *)
PG.Act.AV._6.V_Input.ForceCmd      	   := TRUE;         (* komanda ide na izlaz bez obzira na stanje / alarm *)
PG.Act.AV._6.V_Param.FbOpenExists      := TRUE;         (* postoji DI povratni signal za otvoreni polozaj *)
PG.Act.AV._6.V_Param.FbCloseExists     := TRUE;         (* postoji DI povratni signal za zatvoreni polozaj *)
PG.Act.AV._6.V_Param.OpenMinTime       := T#0s;         (* min vreme drzanja komande otvori pre provere FB *)
PG.Act.AV._6.V_Param.OpenMaxTime       := T#10s;        (* timeout - spring-return brzi od elektromotornog *)
PG.Act.AV._6.V_Param.CloseMinTime      := T#0s;         (* min vreme drzanja komande zatvori pre provere FB *)
PG.Act.AV._6.V_Param.CloseMaxTime      := T#10s;        (* timeout - spring-return brzi od elektromotornog *)
PG.Act.AV._6.V_Param.StableFbDelay     := T#2s;         (* vreme stabilizacije FB signala pre potvrde polozaja *)

(* AV._7: Pneumatski NC leptir ventil DN125 spring-return *)
PG.Act.AV._7.V_Input.Enable            := TRUE;         (* aktivira FB upravljanja ventilom *)
PG.Act.AV._7.V_Input.ForceCmd      	   := TRUE;         (* komanda ide na izlaz bez obzira na stanje / alarm *)
PG.Act.AV._7.V_Param.FbOpenExists      := TRUE;         (* postoji DI povratni signal za otvoreni polozaj *)
PG.Act.AV._7.V_Param.FbCloseExists     := TRUE;         (* postoji DI povratni signal za zatvoreni polozaj *)
PG.Act.AV._7.V_Param.OpenMinTime       := T#0s;         (* min vreme drzanja komande otvori pre provere FB *)
PG.Act.AV._7.V_Param.OpenMaxTime       := T#10s;        (* timeout - spring-return brzi od elektromotornog *)
PG.Act.AV._7.V_Param.CloseMinTime      := T#0s;         (* min vreme drzanja komande zatvori pre provere FB *)
PG.Act.AV._7.V_Param.CloseMaxTime      := T#10s;        (* timeout - spring-return brzi od elektromotornog *)
PG.Act.AV._7.V_Param.StableFbDelay     := T#2s;         (* vreme stabilizacije FB signala pre potvrde polozaja *)

(* -------------------------------------------------------------------------- *)
(* 8) FB_HV_2LS  Rucni leptir ventili RV (_19, _21.._27)                      *)
(* NIOB FLUID 4309 / End Armaturen, rucni C-C sa povratnim signalima.         *)
(* TransitionMaxTime=T#10s: alarm ako tranzicija prekoraci 10s.               *)
(* BothActiveFilterTime=T#500ms: debounce oba krajnja signala.                *)
(* -------------------------------------------------------------------------- *)
(* RV._19: Rucni ventil posle membranskog ventila PG_PV01 *)
PG.Act.RV._19.HV_Input.Enable          := TRUE;         (* aktivira FB monitoringa rucnog ventila *)
PG.Act.RV._19.HV_Param.TransitionMaxTime := T#10s;      (* timeout alarm pri tranziciji polozaja *)
PG.Act.RV._19.HV_Param.BothActiveFilterTime := T#500ms; (* debounce za oba FB aktivna istovremeno *)

(* RV._21: Rucni ventil posle membranskog ventila PG_PV02 *)
PG.Act.RV._21.HV_Input.Enable          := TRUE;         (* aktivira FB monitoringa rucnog ventila *)
PG.Act.RV._21.HV_Param.TransitionMaxTime := T#10s;      (* timeout alarm pri tranziciji polozaja *)
PG.Act.RV._21.HV_Param.BothActiveFilterTime := T#500ms; (* debounce za oba FB aktivna istovremeno *)

(* RV._22: Drenazni total ventil na dnu prihvatnog tanka *)
PG.Act.RV._22.HV_Input.Enable          := TRUE;         (* aktivira FB monitoringa rucnog ventila *)
PG.Act.RV._22.HV_Param.TransitionMaxTime := T#10s;      (* timeout alarm pri tranziciji polozaja *)
PG.Act.RV._22.HV_Param.BothActiveFilterTime := T#500ms; (* debounce za oba FB aktivna istovremeno *)

(* RV._23: Ulaz u Pumpu PG_Pu01 *)
PG.Act.RV._23.HV_Input.Enable          := TRUE;         (* aktivira FB monitoringa rucnog ventila *)
PG.Act.RV._23.HV_Param.TransitionMaxTime := T#10s;      (* timeout alarm pri tranziciji polozaja *)
PG.Act.RV._23.HV_Param.BothActiveFilterTime := T#500ms; (* debounce za oba FB aktivna istovremeno *)

(* RV._24: Ulaz u Pumpu PG_Pu02 *)
PG.Act.RV._24.HV_Input.Enable          := TRUE;         (* aktivira FB monitoringa rucnog ventila *)
PG.Act.RV._24.HV_Param.TransitionMaxTime := T#10s;      (* timeout alarm pri tranziciji polozaja *)
PG.Act.RV._24.HV_Param.BothActiveFilterTime := T#500ms; (* debounce za oba FB aktivna istovremeno *)

(* RV._25: Bajpasni izlaz iz tanka ka instalaciji za izbacivanje gasa van kotlarnice *)
PG.Act.RV._25.HV_Input.Enable          := TRUE;         (* aktivira FB monitoringa rucnog ventila *)
PG.Act.RV._25.HV_Param.TransitionMaxTime := T#10s;      (* timeout alarm pri tranziciji polozaja *)
PG.Act.RV._25.HV_Param.BothActiveFilterTime := T#500ms; (* debounce za oba FB aktivna istovremeno *)

(* RV._26: Ulaz u vakuum pumpu *)
PG.Act.RV._26.HV_Input.Enable          := TRUE;         (* aktivira FB monitoringa rucnog ventila *)
PG.Act.RV._26.HV_Param.TransitionMaxTime := T#10s;      (* timeout alarm pri tranziciji polozaja *)
PG.Act.RV._26.HV_Param.BothActiveFilterTime := T#500ms; (* debounce za oba FB aktivna istovremeno *)

(* RV._27: Izlaz iz vakuum pumpe ka instalaciji za izbacivanje gasa van kotlarnice *)
PG.Act.RV._27.HV_Input.Enable          := TRUE;         (* aktivira FB monitoringa rucnog ventila *)
PG.Act.RV._27.HV_Param.TransitionMaxTime := T#10s;      (* timeout alarm pri tranziciji polozaja *)
PG.Act.RV._27.HV_Param.BothActiveFilterTime := T#500ms; (* debounce za oba FB aktivna istovremeno *)

(* -------------------------------------------------------------------------- *)
(* 9) FB_PvAiAo_Fast  Proporcionalni membranski ventili PV (_1.._5)           *)
(* Burkert, AI povratni signal + AO komanda, 4-20mA, mapirano u IoMap.        *)
(* DeviationOnLimit=8%: alarm ako fizicki polozaj odstupa > 8% od SP.         *)
(* DeviationOffLimit=3%: alarm se gasi kada padne ispod 3% odstupanja.        *)
(* -------------------------------------------------------------------------- *)
(* PV._1: Ulazni regulacioni ventil 1 - prihvatni tank, DN050 NC *)
PG.Act.PV._1.PV_Input.Enable               := TRUE;     (* aktivira FB proporc. ventila *)
PG.Act.PV._1.PV_Input.ForceCmd             := TRUE;     (* komanda ide na izlaz bez obzira na stanje / alarm *)
PG.Act.PV._1.PV_Param.HoldOutputOnFault    := TRUE;     (* zadrzava poslednju AO vrednost pri kvar signalu *)
PG.Act.PV._1.PV_Param.DeviationOnLimit     := 8.0;      (* [%] alarm aktivira se kada odstupanje predje 8% *)
PG.Act.PV._1.PV_Param.DeviationOffLimit    := 3.0;      (* [%] alarm gasi se kada odstupanje padne ispod 3% *)
PG.Act.PV._1.PV_Param.DeviationTime        := T#5s;     (* vreme pre aktiviranja alarma odstupanja *)

(* PV._2: Ulazni regulacioni ventil 2 - prihvatni tank, DN050 NC *)
PG.Act.PV._2.PV_Input.Enable               := TRUE;     (* aktivira FB proporc. ventila *)
PG.Act.PV._2.PV_Input.ForceCmd             := TRUE;     (* komanda ide na izlaz bez obzira na stanje / alarm *)
PG.Act.PV._2.PV_Param.HoldOutputOnFault    := TRUE;     (* zadrzava poslednju AO vrednost pri kvar signalu *)
PG.Act.PV._2.PV_Param.DeviationOnLimit     := 8.0;      (* [%] alarm aktivira se kada odstupanje predje 8% *)
PG.Act.PV._2.PV_Param.DeviationOffLimit    := 3.0;      (* [%] alarm gasi se kada odstupanje padne ispod 3% *)
PG.Act.PV._2.PV_Param.DeviationTime        := T#5s;     (* vreme pre aktiviranja alarma odstupanja *)

(* PV._3: Odzracni ventil na ulazu termalne vode u kotlarnicu, DN025 NC *)
PG.Act.PV._3.PV_Input.Enable               := TRUE;     (* aktivira FB proporc. ventila *)
PG.Act.PV._3.PV_Input.ForceCmd             := TRUE;     (* komanda ide na izlaz bez obzira na stanje / alarm *)
PG.Act.PV._3.PV_Param.HoldOutputOnFault    := TRUE;     (* zadrzava poslednju AO vrednost pri kvar signalu *)
PG.Act.PV._3.PV_Param.DeviationOnLimit     := 8.0;      (* [%] alarm aktivira se kada odstupanje predje 8% *)
PG.Act.PV._3.PV_Param.DeviationOffLimit    := 3.0;      (* [%] alarm gasi se kada odstupanje padne ispod 3% *)
PG.Act.PV._3.PV_Param.DeviationTime        := T#5s;     (* vreme pre aktiviranja alarma odstupanja *)

(* PV._4: Odzracni ventil na ulazu termalne vode u prihvatni tank, DN025 NC *)
PG.Act.PV._4.PV_Input.Enable               := TRUE;     (* aktivira FB proporc. ventila *)
PG.Act.PV._4.PV_Input.ForceCmd             := TRUE;     (* komanda ide na izlaz bez obzira na stanje / alarm *)
PG.Act.PV._4.PV_Param.HoldOutputOnFault    := TRUE;     (* zadrzava poslednju AO vrednost pri kvar signalu *)
PG.Act.PV._4.PV_Param.DeviationOnLimit     := 8.0;      (* [%] alarm aktivira se kada odstupanje predje 8% *)
PG.Act.PV._4.PV_Param.DeviationOffLimit    := 3.0;      (* [%] alarm gasi se kada odstupanje padne ispod 3% *)
PG.Act.PV._4.PV_Param.DeviationTime        := T#5s;     (* vreme pre aktiviranja alarma odstupanja *)

(* PV._5: Dodatni proporcionalni ventil, Fast varijanta kao i ostali PV kanali *)
PG.Act.PV._5.PV_Input.Enable               := TRUE;     (* aktivira FB proporc. ventila *)
PG.Act.PV._5.PV_Input.ForceCmd             := TRUE;     (* komanda ide na izlaz bez obzira na stanje / alarm *)
PG.Act.PV._5.PV_Param.HoldOutputOnFault    := TRUE;     (* zadrzava poslednju AO vrednost pri kvar signalu *)
PG.Act.PV._5.PV_Param.DeviationOnLimit     := 8.0;      (* [%] alarm aktivira se kada odstupanje predje 8% *)
PG.Act.PV._5.PV_Param.DeviationOffLimit    := 3.0;      (* [%] alarm gasi se kada odstupanje padne ispod 3% *)
PG.Act.PV._5.PV_Param.DeviationTime        := T#5s;     (* vreme pre aktiviranja alarma odstupanja *)

(* -------------------------------------------------------------------------- *)
(* 10) vfdMain  Pumpe Pu (_1, _2)  Grundfoss CR45-2A, DIO metod              *)
(* Frekventni opseg: 0-50 Hz. w_run_fwd, w_reset (DO) i w_freq (AO=16bit)   *)
(* mapirani u IoMap. addr_struct se postavlja jednom ovde.                    *)
(* -------------------------------------------------------------------------- *)

(* Pu._1: Pumpa za snabdevanje potrosaca 01, vertikalna visestepena Grundfoss CR45, METOD_DIO *)
PG.Act.Pu._1.settings.METOD_OF_CONTROL          := METOD_DIO;  (* DIO metod: run_fwd/reset/freq kroz IoMap *)
PG.Act.Pu._1.settings.MIN_Freq                  := 0.0;        (* [Hz] minimalna frekvencija - pumpa stoji *)
PG.Act.Pu._1.settings.MAX_Freq                  := 70.0;       (* [Hz] maksimalna frekvencija motora - 50Hz mreza *)
PG.Act.Pu._1.settings.HaveOverCurrentProtection := FALSE;      (* bez hardverske strujne zastite u VFD *)
PG.Act.Pu._1.cmds.Enable                        := TRUE;       (* aktivira VFD upravljanje *)
PG.Act.Pu._1.cmds.en_autoReset                  := TRUE;       (* automatski reset greske frekventnog regulatora *)
PG.Act.Pu.VFD_function._1.addr_struct           := ADR(PG.Act.Pu._1);  (* vezuje vfdMain FB za VFD_type strukturu pumpe *)

(* Pu._2: Pumpa za snabdevanje potrosaca 02, vertikalna visestepena Grundfoss CR45, METOD_DIO *)
PG.Act.Pu._2.settings.METOD_OF_CONTROL          := METOD_DIO;  (* DIO metod: run_fwd/reset/freq kroz IoMap *)
PG.Act.Pu._2.settings.MIN_Freq                  := 0.0;        (* [Hz] minimalna frekvencija - pumpa stoji *)
PG.Act.Pu._2.settings.MAX_Freq                  := 50.0;       (* [Hz] maksimalna frekvencija motora - 50Hz mreza *)
PG.Act.Pu._2.settings.HaveOverCurrentProtection := FALSE;      (* bez hardverske strujne zastite u VFD *)
PG.Act.Pu._2.cmds.Enable                        := TRUE;       (* aktivira VFD upravljanje *)
PG.Act.Pu._2.cmds.en_autoReset                  := TRUE;       (* automatski reset greske frekventnog regulatora *)
PG.Act.Pu.VFD_function._2.addr_struct           := ADR(PG.Act.Pu._2);  (* vezuje vfdMain FB za VFD_type strukturu pumpe *)

END_PROGRAM
```

### Program Logical/DeviceCtrl (IEC)

#### Exit.st - Exit code
```iecst
PROGRAM _EXIT
	(* DeviceCtrl nema resurse koje treba zatvarati. *)
END_PROGRAM
```

#### Variables.var - Local variables
```iecst
VAR
	Pu1_1_plus : BOOL;
	Pu1_01_plus : BOOL;
	Pu1_1_minus : BOOL;
	Pu1_01_minus : BOOL;
	Pu2_1_plus : BOOL;
	Pu2_01_plus : BOOL;
	Pu2_1_minus : BOOL;
	Pu2_01_minus : BOOL;
END_VAR
```

#### CommandMap.st
```iecst
ACTION CommandMap:
	(* ======================================================================== *)
	(* 1) Adapter RETAIN ulaznih ventila                                        *)
	(* ======================================================================== *)
	PG.Act.AV._1.Open := PGRad.CmdRetain.V01_Open;
	PG.Act.AV._2.Open := PGRad.CmdRetain.V02_Open;

	(* ======================================================================== *)
	(* 2) Adapter neretentivnog upravljackog vektora                            *)
	(* ======================================================================== *)
	IF PGRad_Cmd.Aktivan THEN
		PG.Act.AV._3.Open := PGRad_Cmd.Ventili._03_Open;
		PG.Act.AV._4.Open := PGRad_Cmd.Ventili._04_Open;
		PG.Act.AV._5.Open := PGRad_Cmd.Ventili._05_Open;
		PG.Act.AV._6.Open := PGRad_Cmd.Ventili._06_Open;
		PG.Act.AV._7.Open := PGRad_Cmd.Ventili._07_Open;

		PG.Act.PV._1.PV_Input.Enable := PGRad_Cmd.PropVentili.PV01.Enable;
		PG.Act.PV._1.PV_Input.EnableManual := FALSE;
		PG.Act.PV._1.PV_Input.SP_Percent := PGRad_Cmd.PropVentili.PV01.SP_Percent;
		PG.Act.PV._2.PV_Input.Enable := PGRad_Cmd.PropVentili.PV02.Enable;
		PG.Act.PV._2.PV_Input.EnableManual := FALSE;
		PG.Act.PV._2.PV_Input.SP_Percent := PGRad_Cmd.PropVentili.PV02.SP_Percent;
		PG.Act.PV._5.PV_Input.Enable := PGRad_Cmd.PropVentili.PV05.Enable;
		PG.Act.PV._5.PV_Input.EnableManual := FALSE;
		PG.Act.PV._5.PV_Input.SP_Percent := PGRad_Cmd.PropVentili.PV05.SP_Percent;
	END_IF;
END_ACTION
```

#### ValveCtrl.st
```iecst
ACTION ValveCtrl:
	(* ======================================================================== *)
	(* 1) ProcessUnit izlazi odzracnih ventila                                  *)
	(* ======================================================================== *)
	(* ProcessUnit poseduje SP za PV03/PV04; manualni FB ulaz je prisilno iskljucen. *)
	PG.Act.PV._3.PV_Input.EnableManual := FALSE;
	PG.Act.PV._3.PV_Input.SP_Percent := PGRad_AirRelease.PV03.FB.AR_Output.ValveSP_Percent;
	PG.Act.PV._4.PV_Input.EnableManual := FALSE;
	PG.Act.PV._4.PV_Input.SP_Percent := PGRad_AirRelease.PV04.FB.AR_Output.ValveSP_Percent;

	(* ======================================================================== *)
	(* 2) Granice proporcionalnih ventila procesa                               *)
	(* ======================================================================== *)
	(* Clamp 0..100% primenjuje se i na manualnu vrednost i na automatski SP. *)
	IF PG.Act.PV._1.PV_Input.ManualValue_Percent > 100.0 THEN
		PG.Act.PV._1.PV_Input.ManualValue_Percent := 100.0;
	ELSIF PG.Act.PV._1.PV_Input.ManualValue_Percent < 0.0 THEN
		PG.Act.PV._1.PV_Input.ManualValue_Percent := 0.0;
	END_IF;
	IF PG.Act.PV._1.PV_Input.SP_Percent > 100.0 THEN
		PG.Act.PV._1.PV_Input.SP_Percent := 100.0;
	ELSIF PG.Act.PV._1.PV_Input.SP_Percent < 0.0 THEN
		PG.Act.PV._1.PV_Input.SP_Percent := 0.0;
	END_IF;

	IF PG.Act.PV._2.PV_Input.ManualValue_Percent > 100.0 THEN
		PG.Act.PV._2.PV_Input.ManualValue_Percent := 100.0;
	ELSIF PG.Act.PV._2.PV_Input.ManualValue_Percent < 0.0 THEN
		PG.Act.PV._2.PV_Input.ManualValue_Percent := 0.0;
	END_IF;
	IF PG.Act.PV._2.PV_Input.SP_Percent > 100.0 THEN
		PG.Act.PV._2.PV_Input.SP_Percent := 100.0;
	ELSIF PG.Act.PV._2.PV_Input.SP_Percent < 0.0 THEN
		PG.Act.PV._2.PV_Input.SP_Percent := 0.0;
	END_IF;

	IF PG.Act.PV._5.PV_Input.ManualValue_Percent > 100.0 THEN
		PG.Act.PV._5.PV_Input.ManualValue_Percent := 100.0;
	ELSIF PG.Act.PV._5.PV_Input.ManualValue_Percent < 0.0 THEN
		PG.Act.PV._5.PV_Input.ManualValue_Percent := 0.0;
	END_IF;
	IF PG.Act.PV._5.PV_Input.SP_Percent > 100.0 THEN
		PG.Act.PV._5.PV_Input.SP_Percent := 100.0;
	ELSIF PG.Act.PV._5.PV_Input.SP_Percent < 0.0 THEN
		PG.Act.PV._5.PV_Input.SP_Percent := 0.0;
	END_IF;
END_ACTION
```

#### PumpCtrl.st
```iecst
ACTION PumpCtrl:
	(* ======================================================================== *)
	(* 1) Rucna korekcija frekvencije pumpi                                     *)
	(* ======================================================================== *)
	IF NOT PGRad_Cmd.Aktivan THEN
		IF EDGEPOS(Pu1_1_plus) THEN
			PG.Act.Pu._1.params.Freq := PG.Act.Pu._1.params.Freq + 1.0;
		END_IF;
		IF EDGEPOS(Pu1_01_plus) THEN
			PG.Act.Pu._1.params.Freq := PG.Act.Pu._1.params.Freq + 0.1;
		END_IF;
		IF EDGEPOS(Pu1_1_minus) THEN
			PG.Act.Pu._1.params.Freq := PG.Act.Pu._1.params.Freq - 1.0;
		END_IF;
		IF EDGEPOS(Pu1_01_minus) THEN
			PG.Act.Pu._1.params.Freq := PG.Act.Pu._1.params.Freq - 0.1;
		END_IF;

		IF EDGEPOS(Pu2_1_plus) THEN
			PG.Act.Pu._2.params.Freq := PG.Act.Pu._2.params.Freq + 1.0;
		END_IF;
		IF EDGEPOS(Pu2_01_plus) THEN
			PG.Act.Pu._2.params.Freq := PG.Act.Pu._2.params.Freq + 0.1;
		END_IF;
		IF EDGEPOS(Pu2_1_minus) THEN
			PG.Act.Pu._2.params.Freq := PG.Act.Pu._2.params.Freq - 1.0;
		END_IF;
		IF EDGEPOS(Pu2_01_minus) THEN
			PG.Act.Pu._2.params.Freq := PG.Act.Pu._2.params.Freq - 0.1;
		END_IF;
	END_IF;

	(* ======================================================================== *)
	(* 2) Granice frekvencije pumpi                                             *)
	(* ======================================================================== *)
	IF PG.Act.Pu._1.params.Freq > 100.0 THEN
		PG.Act.Pu._1.params.Freq := 100.0;
	ELSIF PG.Act.Pu._1.params.Freq < 10.0 THEN
		PG.Act.Pu._1.params.Freq := 10.0;
	END_IF;
	IF PG.Act.Pu._2.params.Freq > 50.0 THEN
		PG.Act.Pu._2.params.Freq := 50.0;
	ELSIF PG.Act.Pu._2.params.Freq < 10.0 THEN
		PG.Act.Pu._2.params.Freq := 10.0;
	END_IF;
END_ACTION
```
